  MoveL 3672 to (108.07, 245.49, -10) mm, rotated rx 180 ry 0 rz 180 deg; joints [-10.553, -45.82, 118.267, 168.944, 72.753, -176.684]
  MoveL 3673 to (108.64, 236.5, -10) mm, rotated rx -180 ry 0 rz 180 deg; joints [-10.17, -45.837, 118.333, 169.347, 72.78, -176.813]
  MoveL 3674 to (109.78, 227.56, -10) mm, rotated rx 180 ry 0 rz 180 deg; joints [-9.785, -45.844, 118.36, 169.751, 72.778, -176.936]
  MoveL 3675 to (111.49, 218.72, -10) mm, rotated rx -180 ry 0 rz -180 deg; joints [-9.4, -45.841, 118.347, 170.153, 72.749, -177.053]
  MoveL 3676 to (113.75, 209.99, -10) mm, rotated rx 180 ry 0 rz -180 deg; joints [-9.016, -45.827, 118.294, 170.552, 72.691, -177.166]
  MoveL 3677 to (116.56, 201.43, -10) mm, rotated rx 180 ry 0 rz -180 deg; joints [-8.636, -45.803, 118.202, 170.947, 72.605, -177.273]
  MoveL 3678 to (119.91, 193.07, -10) mm, rotated rx -180 ry 0 rz 180 deg; joints [-8.262, -45.769, 118.071, 171.334, 72.492, -177.375]
  MoveL 3679 to (123.79, 184.93, -10) mm, rotated rx 180 ry 0 rz 180 deg; joints [-7.896, -45.724, 117.902, 171.712, 72.352, -177.471]
  MoveL 3680 to (128.17, 177.06, -10) mm, rotated rx -180 ry 0 rz -180 deg; joints [-7.539, -45.669, 117.695, 172.079, 72.186, -177.563]
  MoveL 3681 to (133.04, 169.48, -10) mm, rotated rx 180 ry 0 rz 180 deg; joints [-7.194, -45.604, 117.451, 172.434, 71.995, -177.649]
  MoveL 3682 to (138.38, 162.22, -10) mm, rotated rx -180 ry 0 rz -180 deg; joints [-6.862, -45.529, 117.172, 172.774, 71.779, -177.73]
  MoveL 3683 to (144.17, 155.32, -10) mm, rotated rx -180 ry 0 rz -180 deg; joints [-6.544, -45.444, 116.858, 173.099, 71.54, -177.805]
  MoveL 3684 to (150.39, 148.8, -10) mm, rotated rx 180 ry 0 rz -180 deg; joints [-6.243, -45.349, 116.512, 173.406, 71.279, -177.875]
  MoveL 3685 to (157.01, 142.68, -10) mm, rotated rx 180 ry 0 rz 180 deg; joints [-5.96, -45.245, 116.135, 173.695, 70.998, -177.94]
  MoveL 3686 to (164, 137, -10) mm, rotated rx 180 ry 0 rz -180 deg; joints [-5.695, -45.131, 115.729, 173.964, 70.697, -177.998]
  MoveL 3687 to (171.34, 131.78, -10) mm, rotated rx 180 ry 0 rz -180 deg; joints [-5.45, -45.008, 115.294, 174.212, 70.379, -178.051]
  MoveL 3688 to (179, 127.02, -10) mm, rotated rx 180 ry 0 rz -180 deg; joints [-5.226, -44.877, 114.834, 174.439, 70.045, -178.097]
  MoveL 3689 to (186.94, 122.77, -10) mm, rotated rx -180 ry 0 rz -180 deg; joints [-5.024, -44.737, 114.351, 174.643, 69.696, -178.136]
  MoveL 3690 to (195.14, 119.03, -10) mm, rotated rx 180 ry 0 rz -180 deg; joints [-4.843, -44.589, 113.845, 174.823, 69.334, -178.169]
  MoveL 3691 to (203.56, 115.81, -10) mm, rotated rx 180 ry 0 rz -180 deg; joints [-4.685, -44.433, 113.321, 174.98, 68.961, -178.194]
  MoveL 3692 to (212.16, 113.13, -10) mm, rotated rx -180 ry 0 rz -180 deg; joints [-4.549, -44.271, 112.779, 175.112, 68.579, -178.211]
  MoveL 3693 to (220.92, 111.01, -10) mm, rotated rx -180 ry 0 rz -180 deg; joints [-4.437, -44.102, 112.222, 175.22, 68.189, -178.22]
  MoveL 3694 to (229.79, 109.45, -10) mm, rotated rx 180 ry 0 rz -180 deg; joints [-4.348, -43.927, 111.652, 175.303, 67.792, -178.221]
  MoveL 3695 to (238.75, 108.45, -10) mm, rotated rx -180 ry 0 rz 180 deg; joints [-4.282, -43.747, 111.072, 175.361, 67.392, -178.213]
  MoveL 3696 to (247.75, 108.02, -10) mm, rotated rx 180 ry 0 rz -180 deg; joints [-4.239, -43.563, 110.484, 175.394, 66.988, -178.196]
  MoveL 3697 to (256.76, 108.16, -10) mm, rotated rx -180 ry 0 rz -180 deg; joints [-4.218, -43.375, 109.891, 175.402, 66.584, -178.17]
  MoveL 3698 to (265.74, 108.87, -10) mm, rotated rx 180 ry 0 rz -180 deg; joints [-4.22, -43.183, 109.294, 175.386, 66.179, -178.133]
  MoveL 3699 to (274.66, 110.16, -10) mm, rotated rx 180 ry 0 rz 180 deg; joints [-4.244, -42.99, 108.697, 175.345, 65.778, -178.087]
  MoveL 3700 to (283.48, 112, -10) mm, rotated rx 180 ry 0 rz 180 deg; joints [-4.29, -42.795, 108.101, 175.28, 65.379, -178.03]
  MoveL 3701 to (292.16, 114.4, -10) mm, rotated rx 180 ry 0 rz 180 deg; joints [-4.356, -42.6, 107.508, 175.192, 64.986, -177.963]
  MoveL 3702 to (300.68, 117.35, -10) mm, rotated rx 180 ry 0 rz 180 deg; joints [-4.443, -42.405, 106.922, 175.081, 64.6, -177.886]
  MoveL 3703 to (308.99, 120.83, -10) mm, rotated rx 180 ry 0 rz 180 deg; joints [-4.549, -42.211, 106.345, 174.947, 64.222, -177.798]
  MoveL 3704 to (317.06, 124.83, -10) mm, rotated rx 180 ry 0 rz 180 deg; joints [-4.674, -42.019, 105.778, 174.791, 63.853, -177.7]
  MoveL 3705 to (324.87, 129.34, -10) mm, rotated rx -180 ry 0 rz 180 deg; joints [-4.818, -41.829, 105.224, 174.615, 63.495, -177.591]
  MoveL 3706 to (332.37, 134.33, -10) mm, rotated rx -180 ry 0 rz -180 deg; joints [-4.978, -41.644, 104.684, 174.418, 63.15, -177.473]
  MoveL 3707 to (339.54, 139.79, -10) mm, rotated rx -180 ry 0 rz 180 deg; joints [-5.156, -41.463, 104.162, 174.202, 62.818, -177.344]
  MoveL 3708 to (346.35, 145.69, -10) mm, rotated rx 180 ry 0 rz 180 deg; joints [-5.349, -41.288, 103.659, 173.968, 62.501, -177.206]
  MoveL 3709 to (352.77, 152.01, -10) mm, rotated rx -180 ry 0 rz 180 deg; joints [-5.557, -41.119, 103.176, 173.716, 62.2, -177.06]
  MoveL 3710 to (358.78, 158.72, -10) mm, rotated rx 180 ry 0 rz -180 deg; joints [-5.778, -40.957, 102.717, 173.447, 61.916, -176.905]
  MoveL 3711 to (364.35, 165.81, -10) mm, rotated rx 180 ry 0 rz -180 deg; joints [-6.013, -40.803, 102.282, 173.164, 61.65, -176.742]
  MoveL 3712 to (369.46, 173.23, -10) mm, rotated rx 180 ry 0 rz 180 deg; joints [-6.26, -40.657, 101.873, 172.866, 61.403, -176.572]
  MoveL 3713 to (374.09, 180.96, -10) mm, rotated rx 180 ry 0 rz 180 deg; joints [-6.518, -40.521, 101.491, 172.555, 61.176, -176.395]
  MoveL 3714 to (378.22, 188.97, -10) mm, rotated rx -180 ry 0 rz 180 deg; joints [-6.787, -40.394, 101.139, 172.233, 60.97, -176.213]
  MoveL 3715 to (381.83, 197.22, -10) mm, rotated rx 180 ry 0 rz -180 deg; joints [-7.064, -40.278, 100.818, 171.9, 60.785, -176.026]
  MoveL 3716 to (384.91, 205.69, -10) mm, rotated rx -180 ry 0 rz 180 deg; joints [-7.35, -40.174, 100.528, 171.558, 60.622, -175.836]
  MoveL 3717 to (387.45, 214.34, -10) mm, rotated rx 180 ry 0 rz 180 deg; joints [-7.643, -40.08, 100.271, 171.208, 60.482, -175.642]
  MoveL 3718 to (389.43, 223.13, -10) mm, rotated rx -180 ry 0 rz -180 deg; joints [-7.943, -39.999, 100.048, 170.852, 60.365, -175.447]
  MoveL 3719 to (390.86, 232.02, -10) mm, rotated rx -180 ry 0 rz -180 deg; joints [-8.248, -39.931, 99.86, 170.491, 60.272, -175.252]
  MoveL 3720 to (391.71, 240.99, -10) mm, rotated rx -180 ry 0 rz -180 deg; joints [-8.558, -39.875, 99.707, 170.126, 60.202, -175.056]
  MoveL 3721 to (392, 250, -10) mm, rotated rx 180 ry 0 rz -180 deg; joints [-8.871, -39.832, 99.591, 169.759, 60.157, -174.863]
  MoveL 3722 to (380, 250, -10) mm, rotated rx -180 ry 0 rz 180 deg; joints [-8.937, -40.137, 100.428, 169.737, 60.687, -174.934]
  MoveL 3723 to (379.74, 258.25, -10) mm, rotated rx 180 ry 0 rz 180 deg; joints [-9.229, -40.111, 100.355, 169.4, 60.667, -174.762]
  MoveL 3724 to (378.95, 266.46, -10) mm, rotated rx 180 ry 0 rz -180 deg; joints [-9.521, -40.096, 100.315, 169.063, 60.669, -174.592]
  MoveL 3725 to (377.65, 274.6, -10) mm, rotated rx 180 ry 0 rz 180 deg; joints [-9.815, -40.094, 100.309, 168.727, 60.694, -174.428]
  MoveL 3726 to (375.83, 282.65, -10) mm, rotated rx 180 ry 0 rz -180 deg; joints [-10.108, -40.104, 100.337, 168.395, 60.74, -174.268]
  MoveL 3727 to (373.51, 290.56, -10) mm, rotated rx -180 ry 0 rz -180 deg; joints [-10.4, -40.127, 100.399, 168.067, 60.808, -174.115]
  MoveL 3728 to (370.69, 298.32, -10) mm, rotated rx 180 ry 0 rz -180 deg; joints [-10.689, -40.161, 100.495, 167.744, 60.898, -173.969]
  MoveL 3729 to (367.38, 305.87, -10) mm, rotated rx 180 ry 0 rz 180 deg; joints [-10.976, -40.208, 100.623, 167.427, 61.009, -173.831]
  MoveL 3730 to (363.6, 313.21, -10) mm, rotated rx 180 ry 0 rz 180 deg; joints [-11.259, -40.266, 100.785, 167.119, 61.14, -173.701]
  MoveL 3731 to (359.36, 320.28, -10) mm, rotated rx 180 ry 0 rz 180 deg; joints [-11.537, -40.336, 100.978, 166.819, 61.291, -173.581]
  MoveL 3732 to (354.69, 327.08, -10) mm, rotated rx 180 ry 0 rz -180 deg; joints [-11.809, -40.417, 101.203, 166.529, 61.462, -173.471]
  MoveL 3733 to (349.59, 333.56, -10) mm, rotated rx -180 ry 0 rz -180 deg; joints [-12.075, -40.509, 101.458, 166.25, 61.651, -173.372]
  MoveL 3734 to (344.09, 339.71, -10) mm, rotated rx 180 ry 0 rz 180 deg; joints [-12.333, -40.611, 101.743, 165.982, 61.859, -173.284]
  MoveL 3735 to (338.21, 345.5, -10) mm, rotated rx -180 ry 0 rz 180 deg; joints [-12.582, -40.722, 102.056, 165.728, 62.083, -173.208]
  MoveL 3736 to (331.97, 350.9, -10) mm, rotated rx -180 ry 0 rz -180 deg; joints [-12.823, -40.843, 102.397, 165.487, 62.324, -173.144]
  MoveL 3737 to (325.41, 355.89, -10) mm, rotated rx 180 ry 0 rz 180 deg; joints [-13.053, -40.973, 102.763, 165.26, 62.581, -173.092]
  MoveL 3738 to (318.54, 360.46, -10) mm, rotated rx -180 ry 0 rz 180 deg; joints [-13.272, -41.111, 103.154, 165.049, 62.852, -173.053]
  MoveL 3739 to (311.4, 364.59, -10) mm, rotated rx 180 ry 0 rz -180 deg; joints [-13.479, -41.256, 103.567, 164.854, 63.136, -173.027]
  MoveL 3740 to (304, 368.25, -10) mm, rotated rx -180 ry 0 rz 180 deg; joints [-13.673, -41.408, 104.003, 164.675, 63.433, -173.013]
  MoveL 3741 to (296.4, 371.44, -10) mm, rotated rx -180 ry 0 rz -180 deg; joints [-13.854, -41.566, 104.457, 164.514, 63.742, -173.012]
  MoveL 3742 to (288.6, 374.14, -10) mm, rotated rx -180 ry 0 rz 180 deg; joints [-14.02, -41.729, 104.93, 164.371, 64.06, -173.023]
  MoveL 3743 to (280.65, 376.34, -10) mm, rotated rx -180 ry 0 rz -180 deg; joints [-14.172, -41.896, 105.419, 164.246, 64.388, -173.047]
  MoveL 3744 to (272.57, 378.03, -10) mm, rotated rx 180 ry 0 rz 180 deg; joints [-14.307, -42.068, 105.923, 164.14, 64.724, -173.084]
  MoveL 3745 to (264.41, 379.2, -10) mm, rotated rx 180 ry 0 rz -180 deg; joints [-14.426, -42.242, 106.439, 164.054, 65.067, -173.132]
  MoveL 3746 to (256.19, 379.85, -10) mm, rotated rx -180 ry 0 rz 180 deg; joints [-14.527, -42.419, 106.965, 163.987, 65.415, -173.191]
  MoveL 3747 to (247.94, 379.98, -10) mm, rotated rx -180 ry 0 rz 180 deg; joints [-14.611, -42.597, 107.499, 163.941, 65.767, -173.262]
  MoveL 3748 to (239.7, 379.59, -10) mm, rotated rx -180 ry 0 rz -180 deg; joints [-14.676, -42.775, 108.04, 163.915, 66.123, -173.343]
  MoveL 3749 to (231.5, 378.68, -10) mm, rotated rx -180 ry 0 rz -180 deg; joints [-14.722, -42.954, 108.585, 163.91, 66.48, -173.434]
  MoveL 3750 to (223.38, 377.24, -10) mm, rotated rx -180 ry 0 rz 180 deg; joints [-14.748, -43.131, 109.132, 163.926, 66.838, -173.534]
  MoveL 3751 to (215.36, 375.3, -10) mm, rotated rx -180 ry 0 rz -180 deg; joints [-14.754, -43.307, 109.679, 163.962, 67.196, -173.643]
  MoveL 3752 to (207.48, 372.85, -10) mm, rotated rx 180 ry 0 rz 180 deg; joints [-14.74, -43.48, 110.223, 164.02, 67.551, -173.759]
  MoveL 3753 to (199.78, 369.91, -10) mm, rotated rx -180 ry 0 rz -180 deg; joints [-14.705, -43.651, 110.763, 164.099, 67.903, -173.883]
  MoveL 3754 to (192.27, 366.48, -10) mm, rotated rx -180 ry 0 rz -180 deg; joints [-14.649, -43.817, 111.296, 164.199, 68.25, -174.014]
  MoveL 3755 to (185, 362.58, -10) mm, rotated rx 180 ry 0 rz -180 deg; joints [-14.573, -43.979, 111.821, 164.32, 68.59, -174.15]
  MoveL 3756 to (177.99, 358.23, -10) mm, rotated rx 180 ry 0 rz -180 deg; joints [-14.475, -44.136, 112.335, 164.462, 68.924, -174.29]
  MoveL 3757 to (171.27, 353.45, -10) mm, rotated rx -180 ry 0 rz -180 deg; joints [-14.356, -44.288, 112.835, 164.624, 69.249, -174.435]
  MoveL 3758 to (164.87, 348.25, -10) mm, rotated rx -180 ry 0 rz 180 deg; joints [-14.217, -44.433, 113.32, 164.806, 69.563, -174.583]
  MoveL 3759 to (158.81, 342.65, -10) mm, rotated rx -180 ry 0 rz -180 deg; joints [-14.057, -44.572, 113.789, 165.007, 69.866, -174.733]
  MoveL 3760 to (153.12, 336.68, -10) mm, rotated rx -180 ry 0 rz 180 deg; joints [-13.877, -44.704, 114.237, 165.228, 70.157, -174.885]
  MoveL 3761 to (147.81, 330.36, -10) mm, rotated rx 180 ry 0 rz 180 deg; joints [-13.677, -44.828, 114.665, 165.466, 70.433, -175.038]
  MoveL 3762 to (142.92, 323.72, -10) mm, rotated rx 180 ry 0 rz 180 deg; joints [-13.459, -44.944, 115.07, 165.722, 70.694, -175.191]
  MoveL 3763 to (138.46, 316.78, -10) mm, rotated rx 180 ry 0 rz 180 deg; joints [-13.223, -45.052, 115.45, 165.995, 70.938, -175.343]
  MoveL 3764 to (134.45, 309.57, -10) mm, rotated rx 180 ry 0 rz -180 deg; joints [-12.97, -45.152, 115.804, 166.283, 71.164, -175.494]
  MoveL 3765 to (130.91, 302.12, -10) mm, rotated rx -180 ry 0 rz -180 deg; joints [-12.7, -45.243, 116.13, 166.585, 71.371, -175.643]
  MoveL 3766 to (127.84, 294.46, -10) mm, rotated rx -180 ry 0 rz -180 deg; joints [-12.416, -45.325, 116.426, 166.901, 71.559, -175.79]
  MoveL 3767 to (125.27, 286.63, -10) mm, rotated rx -180 ry 0 rz -180 deg; joints [-12.118, -45.398, 116.691, 167.228, 71.725, -175.934]
  MoveL 3768 to (123.19, 278.64, -10) mm, rotated rx 180 ry 0 rz 180 deg; joints [-11.808, -45.462, 116.925, 167.566, 71.869, -176.075]
  MoveL 3769 to (121.63, 270.54, -10) mm, rotated rx 180 ry 0 rz -180 deg; joints [-11.487, -45.516, 117.125, 167.913, 71.99, -176.212]
  MoveL 3770 to (120.59, 262.36, -10) mm, rotated rx 180 ry 0 rz 180 deg; joints [-11.157, -45.561, 117.292, 168.267, 72.087, -176.345]
  MoveL 3771 to (120.07, 254.12, -10) mm, rotated rx 180 ry 0 rz 180 deg; joints [-10.819, -45.597, 117.423, 168.627, 72.161, -176.474]
  MoveL 3772 to (120.07, 245.88, -10) mm, rotated rx -180 ry 0 rz -180 deg; joints [-10.476, -45.622, 117.519, 168.992, 72.209, -176.598]
  MoveL 3773 to (120.59, 237.64, -10) mm, rotated rx 180 ry 0 rz -180 deg; joints [-10.128, -45.638, 117.58, 169.358, 72.232, -176.718]
  MoveL 3774 to (121.63, 229.46, -10) mm, rotated rx 180 ry 0 rz -180 deg; joints [-9.779, -45.645, 117.604, 169.726, 72.23, -176.834]
  MoveL 3775 to (123.19, 221.36, -10) mm, rotated rx 180 ry 0 rz 180 deg; joints [-9.429, -45.642, 117.592, 170.092, 72.203, -176.944]
  MoveL 3776 to (125.27, 213.37, -10) mm, rotated rx -180 ry 0 rz 180 deg; joints [-9.081, -45.629, 117.544, 170.455, 72.15, -177.05]
  MoveL 3777 to (127.84, 205.54, -10) mm, rotated rx -180 ry 0 rz -180 deg; joints [-8.736, -45.607, 117.46, 170.814, 72.072, -177.15]
  MoveL 3778 to (130.91, 197.88, -10) mm, rotated rx 180 ry 0 rz -180 deg; joints [-8.396, -45.574, 117.341, 171.166, 71.969, -177.246]
  MoveL 3779 to (134.45, 190.43, -10) mm, rotated rx -180 ry 0 rz -180 deg; joints [-8.064, -45.533, 117.186, 171.511, 71.841, -177.337]
  MoveL 3780 to (138.46, 183.22, -10) mm, rotated rx -180 ry 0 rz 180 deg; joints [-7.739, -45.482, 116.998, 171.845, 71.69, -177.422]
  MoveL 3781 to (142.92, 176.28, -10) mm, rotated rx 180 ry 0 rz 180 deg; joints [-7.425, -45.421, 116.776, 172.168, 71.516, -177.503]
  MoveL 3782 to (147.81, 169.64, -10) mm, rotated rx -180 ry 0 rz -180 deg; joints [-7.123, -45.351, 116.521, 172.479, 71.32, -177.579]
  MoveL 3783 to (153.12, 163.32, -10) mm, rotated rx 180 ry 0 rz 180 deg; joints [-6.834, -45.272, 116.235, 172.775, 71.103, -177.649]
  MoveL 3784 to (158.81, 157.35, -10) mm, rotated rx -180 ry 0 rz 180 deg; joints [-6.559, -45.185, 115.92, 173.056, 70.866, -177.714]
  MoveL 3785 to (164.87, 151.75, -10) mm, rotated rx -180 ry 0 rz 180 deg; joints [-6.3, -45.088, 115.575, 173.32, 70.61, -177.773]
  MoveL 3786 to (171.27, 146.55, -10) mm, rotated rx -180 ry 0 rz 180 deg; joints [-6.058, -44.983, 115.204, 173.566, 70.337, -177.827]
  MoveL 3787 to (177.99, 141.77, -10) mm, rotated rx 180 ry 0 rz 180 deg; joints [-5.833, -44.869, 114.808, 173.793, 70.047, -177.875]
  MoveL 3788 to (185, 137.42, -10) mm, rotated rx 180 ry 0 rz -180 deg; joints [-5.627, -44.747, 114.388, 174.001, 69.743, -177.916]
  MoveL 3789 to (192.27, 133.52, -10) mm, rotated rx -180 ry 0 rz 180 deg; joints [-5.44, -44.618, 113.946, 174.188, 69.425, -177.951]
  MoveL 3790 to (199.78, 130.09, -10) mm, rotated rx -180 ry 0 rz 180 deg; joints [-5.273, -44.482, 113.484, 174.354, 69.095, -177.98]
  MoveL 3791 to (207.48, 127.15, -10) mm, rotated rx 180 ry 0 rz 180 deg; joints [-5.127, -44.339, 113.004, 174.498, 68.755, -178.001]
  MoveL 3792 to (215.36, 124.7, -10) mm, rotated rx -180 ry 0 rz -180 deg; joints [-5.001, -44.189, 112.509, 174.62, 68.406, -178.015]
  MoveL 3793 to (223.38, 122.76, -10) mm, rotated rx 180 ry 0 rz 180 deg; joints [-4.896, -44.034, 112, 174.72, 68.05, -178.022]
  MoveL 3794 to (231.5, 121.32, -10) mm, rotated rx -180 ry 0 rz 180 deg; joints [-4.812, -43.874, 111.479, 174.798, 67.688, -178.02]
  MoveL 3795 to (239.7, 120.41, -10) mm, rotated rx 180 ry 0 rz 180 deg; joints [-4.749, -43.709, 110.948, 174.852, 67.322, -178.011]
  MoveL 3796 to (247.94, 120.02, -10) mm, rotated rx -180 ry 0 rz 180 deg; joints [-4.707, -43.539, 110.41, 174.884, 66.953, -177.993]
  MoveL 3797 to (256.19, 120.15, -10) mm, rotated rx 180 ry 0 rz -180 deg; joints [-4.686, -43.367, 109.867, 174.893, 66.583, -177.966]
  MoveL 3798 to (264.41, 120.8, -10) mm, rotated rx 180 ry 0 rz 180 deg; joints [-4.685, -43.192, 109.321, 174.879, 66.213, -177.93]
  MoveL 3799 to (272.57, 121.98, -10) mm, rotated rx -180 ry 0 rz 180 deg; joints [-4.704, -43.015, 108.774, 174.843, 65.845, -177.885]
  MoveL 3800 to (280.65, 123.66, -10) mm, rotated rx 180 ry 0 rz 180 deg; joints [-4.743, -42.837, 108.228, 174.785, 65.481, -177.831]
  MoveL 3801 to (288.6, 125.86, -10) mm, rotated rx -180 ry 0 rz -180 deg; joints [-4.802, -42.658, 107.685, 174.706, 65.121, -177.767]
  MoveL 3802 to (296.4, 128.56, -10) mm, rotated rx -180 ry 0 rz -180 deg; joints [-4.879, -42.48, 107.148, 174.605, 64.767, -177.694]
  MoveL 3803 to (304, 131.75, -10) mm, rotated rx -180 ry 0 rz 180 deg; joints [-4.974, -42.303, 106.619, 174.484, 64.42, -177.612]
  MoveL 3804 to (311.4, 135.41, -10) mm, rotated rx -180 ry 0 rz 180 deg; joints [-5.087, -42.128, 106.1, 174.342, 64.082, -177.521]
  MoveL 3805 to (318.54, 139.54, -10) mm, rotated rx 180 ry 0 rz 180 deg; joints [-5.217, -41.955, 105.592, 174.181, 63.754, -177.42]
  MoveL 3806 to (325.41, 144.11, -10) mm, rotated rx -180 ry 0 rz -180 deg; joints [-5.363, -41.786, 105.097, 174.002, 63.437, -177.31]
  MoveL 3807 to (331.97, 149.1, -10) mm, rotated rx 180 ry 0 rz 180 deg; joints [-5.524, -41.621, 104.619, 173.805, 63.133, -177.192]
  MoveL 3808 to (338.21, 154.5, -10) mm, rotated rx 180 ry 0 rz 180 deg; joints [-5.7, -41.462, 104.157, 173.591, 62.842, -177.065]
  MoveL 3809 to (344.09, 160.29, -10) mm, rotated rx 180 ry 0 rz -180 deg; joints [-5.89, -41.308, 103.715, 173.361, 62.566, -176.93]
  MoveL 3810 to (349.59, 166.44, -10) mm, rotated rx -180 ry 0 rz 180 deg; joints [-6.093, -41.16, 103.294, 173.115, 62.305, -176.788]
  MoveL 3811 to (354.69, 172.92, -10) mm, rotated rx -180 ry 0 rz 180 deg; joints [-6.308, -41.02, 102.895, 172.856, 62.06, -176.639]
  MoveL 3812 to (359.36, 179.72, -10) mm, rotated rx 180 ry 0 rz -180 deg; joints [-6.534, -40.887, 102.52, 172.584, 61.834, -176.484]
  MoveL 3813 to (363.6, 186.79, -10) mm, rotated rx -180 ry 0 rz -180 deg; joints [-6.771, -40.763, 102.171, 172.299, 61.625, -176.323]
  MoveL 3814 to (367.38, 194.13, -10) mm, rotated rx -180 ry 0 rz 180 deg; joints [-7.017, -40.648, 101.848, 172.004, 61.435, -176.158]
  MoveL 3815 to (370.69, 201.68, -10) mm, rotated rx -180 ry 0 rz -180 deg; joints [-7.273, -40.543, 101.553, 171.699, 61.265, -175.988]
  MoveL 3816 to (373.51, 209.44, -10) mm, rotated rx 180 ry 0 rz -180 deg; joints [-7.536, -40.448, 101.288, 171.386, 61.116, -175.815]
  MoveL 3817 to (375.83, 217.35, -10) mm, rotated rx 180 ry 0 rz 180 deg; joints [-7.806, -40.363, 101.052, 171.066, 60.987, -175.64]
  MoveL 3818 to (377.65, 225.4, -10) mm, rotated rx -180 ry 0 rz 180 deg; joints [-8.082, -40.289, 100.848, 170.739, 60.879, -175.463]
  MoveL 3819 to (378.95, 233.54, -10) mm, rotated rx -180 ry 0 rz -180 deg; joints [-8.363, -40.227, 100.675, 170.408, 60.793, -175.286]
  MoveL 3820 to (379.74, 241.75, -10) mm, rotated rx 180 ry 0 rz -180 deg; joints [-8.648, -40.176, 100.535, 170.074, 60.729, -175.109]
  MoveL 3821 to (380, 250, -10) mm, rotated rx -180 ry 0 rz 180 deg; joints [-8.937, -40.137, 100.428, 169.737, 60.687, -174.934]
  MoveL 3822 to (368, 250, -10) mm, rotated rx -180 ry 0 rz 180 deg; joints [-9.004, -40.438, 101.261, 169.714, 61.216, -175.006]
  MoveL 3823 to (367.76, 257.48, -10) mm, rotated rx 180 ry 0 rz 180 deg; joints [-9.27, -40.414, 101.194, 169.407, 61.198, -174.851]
  MoveL 3824 to (367.05, 264.94, -10) mm, rotated rx 180 ry 0 rz 180 deg; joints [-9.538, -40.401, 101.158, 169.1, 61.199, -174.7]
  MoveL 3825 to (365.87, 272.33, -10) mm, rotated rx 180 ry 0 rz 180 deg; joints [-9.806, -40.399, 101.153, 168.795, 61.221, -174.552]
  MoveL 3826 to (364.22, 279.64, -10) mm, rotated rx -180 ry 0 rz 180 deg; joints [-10.075, -40.408, 101.178, 168.492, 61.263, -174.409]
  MoveL 3827 to (362.11, 286.82, -10) mm, rotated rx 180 ry 0 rz -180 deg; joints [-10.341, -40.428, 101.234, 168.193, 61.325, -174.272]
  MoveL 3828 to (359.55, 293.86, -10) mm, rotated rx 180 ry 0 rz -180 deg; joints [-10.606, -40.46, 101.321, 167.899, 61.406, -174.141]
  MoveL 3829 to (356.55, 300.72, -10) mm, rotated rx -180 ry 0 rz 180 deg; joints [-10.868, -40.502, 101.438, 167.611, 61.506, -174.018]
  MoveL 3830 to (353.11, 307.37, -10) mm, rotated rx 180 ry 0 rz 180 deg; joints [-11.127, -40.554, 101.585, 167.33, 61.625, -173.902]
  MoveL 3831 to (349.27, 313.8, -10) mm, rotated rx 180 ry 0 rz 180 deg; joints [-11.381, -40.617, 101.761, 167.057, 61.763, -173.794]
  MoveL 3832 to (345.02, 319.96, -10) mm, rotated rx -180 ry 0 rz -180 deg; joints [-11.629, -40.69, 101.965, 166.793, 61.918, -173.696]
  MoveL 3833 to (340.39, 325.85, -10) mm, rotated rx 180 ry 0 rz 180 deg; joints [-11.871, -40.773, 102.197, 166.538, 62.09, -173.607]
  MoveL 3834 to (335.4, 331.43, -10) mm, rotated rx 180 ry 0 rz -180 deg; joints [-12.107, -40.865, 102.456, 166.295, 62.278, -173.528]
  MoveL 3835 to (330.06, 336.68, -10) mm, rotated rx 180 ry 0 rz 180 deg; joints [-12.334, -40.965, 102.741, 166.063, 62.483, -173.459]
  MoveL 3836 to (324.41, 341.59, -10) mm, rotated rx -180 ry 0 rz -180 deg; joints [-12.553, -41.074, 103.05, 165.843, 62.702, -173.401]
  MoveL 3837 to (318.45, 346.12, -10) mm, rotated rx -180 ry 0 rz 180 deg; joints [-12.762, -41.191, 103.383, 165.637, 62.936, -173.354]
  MoveL 3838 to (312.21, 350.27, -10) mm, rotated rx 180 ry 0 rz -180 deg; joints [-12.961, -41.316, 103.738, 165.445, 63.182, -173.319]
  MoveL 3839 to (305.73, 354.01, -10) mm, rotated rx -180 ry 0 rz -180 deg; joints [-13.149, -41.447, 104.114, 165.267, 63.441, -173.294]
  MoveL 3840 to (299.02, 357.34, -10) mm, rotated rx 180 ry 0 rz 180 deg; joints [-13.325, -41.584, 104.51, 165.104, 63.712, -173.281]
  MoveL 3841 to (292.11, 360.23, -10) mm, rotated rx 180 ry 0 rz 180 deg; joints [-13.488, -41.726, 104.923, 164.958, 63.992, -173.279]
  MoveL 3842 to (285.04, 362.68, -10) mm, rotated rx 180 ry 0 rz -180 deg; joints [-13.639, -41.874, 105.353, 164.828, 64.283, -173.289]
  MoveL 3843 to (277.82, 364.67, -10) mm, rotated rx 180 ry 0 rz 180 deg; joints [-13.775, -42.025, 105.797, 164.715, 64.581, -173.309]
  MoveL 3844 to (270.49, 366.21, -10) mm, rotated rx 180 ry 0 rz -180 deg; joints [-13.896, -42.18, 106.255, 164.619, 64.887, -173.341]
  MoveL 3845 to (263.08, 367.27, -10) mm, rotated rx 180 ry 0 rz -180 deg; joints [-14.002, -42.338, 106.723, 164.541, 65.199, -173.383]
  MoveL 3846 to (255.61, 367.87, -10) mm, rotated rx 180 ry 0 rz 180 deg; joints [-14.093, -42.498, 107.201, 164.481, 65.516, -173.435]
  MoveL 3847 to (248.13, 367.99, -10) mm, rotated rx -180 ry 0 rz -180 deg; joints [-14.167, -42.659, 107.687, 164.44, 65.837, -173.497]
  MoveL 3848 to (240.65, 367.63, -10) mm, rotated rx -180 ry 0 rz -180 deg; joints [-14.224, -42.821, 108.178, 164.418, 66.161, -173.569]
  MoveL 3849 to (233.21, 366.8, -10) mm, rotated rx -180 ry 0 rz -180 deg; joints [-14.263, -42.982, 108.673, 164.414, 66.486, -173.65]
  MoveL 3850 to (225.83, 365.5, -10) mm, rotated rx 180 ry 0 rz -180 deg; joints [-14.284, -43.143, 109.169, 164.43, 66.811, -173.739]
  MoveL 3851 to (218.56, 363.73, -10) mm, rotated rx -180 ry 0 rz 180 deg; joints [-14.288, -43.303, 109.666, 164.464, 67.136, -173.835]
  MoveL 3852 to (211.41, 361.51, -10) mm, rotated rx 180 ry 0 rz 180 deg; joints [-14.273, -43.46, 110.16, 164.519, 67.459, -173.939]
  MoveL 3853 to (204.41, 358.84, -10) mm, rotated rx -180 ry 0 rz -180 deg; joints [-14.239, -43.615, 110.65, 164.592, 67.779, -174.05]
  MoveL 3854 to (197.6, 355.73, -10) mm, rotated rx -180 ry 0 rz -180 deg; joints [-14.186, -43.766, 111.134, 164.684, 68.094, -174.166]
  MoveL 3855 to (191, 352.19, -10) mm, rotated rx 180 ry 0 rz 180 deg; joints [-14.114, -43.914, 111.609, 164.796, 68.403, -174.288]
  MoveL 3856 to (184.64, 348.24, -10) mm, rotated rx 180 ry 0 rz 180 deg; joints [-14.023, -44.057, 112.075, 164.926, 68.705, -174.414]
  MoveL 3857 to (178.54, 343.9, -10) mm, rotated rx -180 ry 0 rz -180 deg; joints [-13.913, -44.195, 112.529, 165.074, 69, -174.543]
  MoveL 3858 to (172.73, 339.18, -10) mm, rotated rx 180 ry 0 rz 180 deg; joints [-13.785, -44.328, 112.969, 165.241, 69.285, -174.676]
  MoveL 3859 to (167.23, 334.1, -10) mm, rotated rx 180 ry 0 rz 180 deg; joints [-13.639, -44.455, 113.393, 165.425, 69.559, -174.811]
  MoveL 3860 to (162.06, 328.68, -10) mm, rotated rx -180 ry 0 rz 180 deg; joints [-13.474, -44.575, 113.799, 165.626, 69.821, -174.948]
  MoveL 3861 to (157.25, 322.94, -10) mm, rotated rx 180 ry 0 rz -180 deg; joints [-13.292, -44.689, 114.187, 165.844, 70.071, -175.086]
  MoveL 3862 to (152.81, 316.91, -10) mm, rotated rx -180 ry 0 rz 180 deg; joints [-13.094, -44.796, 114.553, 166.077, 70.306, -175.224]
  MoveL 3863 to (148.76, 310.61, -10) mm, rotated rx -180 ry 0 rz 180 deg; joints [-12.879, -44.895, 114.897, 166.324, 70.526, -175.362]
  MoveL 3864 to (145.12, 304.07, -10) mm, rotated rx 180 ry 0 rz 180 deg; joints [-12.65, -44.986, 115.217, 166.586, 70.73, -175.5]
  MoveL 3865 to (141.9, 297.31, -10) mm, rotated rx 180 ry 0 rz 180 deg; joints [-12.406, -45.07, 115.512, 166.86, 70.917, -175.636]
  MoveL 3866 to (139.12, 290.36, -10) mm, rotated rx 180 ry 0 rz -180 deg; joints [-12.149, -45.145, 115.78, 167.146, 71.085, -175.77]
  MoveL 3867 to (136.78, 283.24, -10) mm, rotated rx 180 ry 0 rz 180 deg; joints [-11.879, -45.213, 116.02, 167.443, 71.234, -175.901]
  MoveL 3868 to (134.9, 276, -10) mm, rotated rx -180 ry 0 rz -180 deg; joints [-11.6, -45.271, 116.231, 167.749, 71.363, -176.03]
  MoveL 3869 to (133.48, 268.64, -10) mm, rotated rx 180 ry 0 rz 180 deg; joints [-11.31, -45.321, 116.412, 168.063, 71.471, -176.156]
  MoveL 3870 to (132.53, 261.22, -10) mm, rotated rx -180 ry 0 rz 180 deg; joints [-11.013, -45.363, 116.563, 168.383, 71.559, -176.279]
  MoveL 3871 to (132.06, 253.74, -10) mm, rotated rx 180 ry 0 rz -180 deg; joints [-10.709, -45.396, 116.682, 168.708, 71.624, -176.398]
  MoveL 3872 to (132.06, 246.26, -10) mm, rotated rx 180 ry 0 rz 180 deg; joints [-10.4, -45.419, 116.769, 169.037, 71.667, -176.513]
  MoveL 3873 to (132.53, 238.78, -10) mm, rotated rx -180 ry 0 rz -180 deg; joints [-10.087, -45.434, 116.823, 169.368, 71.687, -176.624]
  MoveL 3874 to (133.48, 231.36, -10) mm, rotated rx 180 ry 0 rz 180 deg; joints [-9.773, -45.44, 116.845, 169.7, 71.684, -176.731]
  MoveL 3875 to (134.9, 224, -10) mm, rotated rx -180 ry 0 rz -180 deg; joints [-9.458, -45.437, 116.835, 170.03, 71.659, -176.834]
  MoveL 3876 to (136.78, 216.76, -10) mm, rotated rx 180 ry 0 rz -180 deg; joints [-9.145, -45.426, 116.791, 170.358, 71.611, -176.932]
  MoveL 3877 to (139.12, 209.64, -10) mm, rotated rx -180 ry 0 rz -180 deg; joints [-8.835, -45.405, 116.715, 170.682, 71.54, -177.026]
  MoveL 3878 to (141.9, 202.69, -10) mm, rotated rx 180 ry 0 rz 180 deg; joints [-8.529, -45.375, 116.607, 171, 71.447, -177.115]
  MoveL 3879 to (145.12, 195.93, -10) mm, rotated rx 180 ry 0 rz 180 deg; joints [-8.229, -45.337, 116.468, 171.311, 71.332, -177.199]
  MoveL 3880 to (148.76, 189.39, -10) mm, rotated rx -180 ry 0 rz -180 deg; joints [-7.937, -45.29, 116.297, 171.613, 71.196, -177.279]
  MoveL 3881 to (152.81, 183.09, -10) mm, rotated rx -180 ry 0 rz -180 deg; joints [-7.653, -45.234, 116.096, 171.905, 71.039, -177.354]
  MoveL 3882 to (157.25, 177.06, -10) mm, rotated rx -180 ry 0 rz -180 deg; joints [-7.38, -45.17, 115.866, 172.185, 70.863, -177.424]
  MoveL 3883 to (162.06, 171.32, -10) mm, rotated rx 180 ry 0 rz -180 deg; joints [-7.119, -45.097, 115.608, 172.453, 70.667, -177.489]
  MoveL 3884 to (167.23, 165.9, -10) mm, rotated rx -180 ry 0 rz -180 deg; joints [-6.87, -45.016, 115.322, 172.707, 70.453, -177.548]
  MoveL 3885 to (172.73, 160.82, -10) mm, rotated rx -180 ry 0 rz 180 deg; joints [-6.636, -44.927, 115.011, 172.946, 70.222, -177.603]
  MoveL 3886 to (178.54, 156.1, -10) mm, rotated rx -180 ry 0 rz 180 deg; joints [-6.416, -44.831, 114.675, 173.17, 69.976, -177.651]
  MoveL 3887 to (184.64, 151.76, -10) mm, rotated rx -180 ry 0 rz 180 deg; joints [-6.212, -44.727, 114.316, 173.376, 69.714, -177.694]
  MoveL 3888 to (191, 147.81, -10) mm, rotated rx 180 ry 0 rz 180 deg; joints [-6.024, -44.615, 113.935, 173.565, 69.439, -177.732]
  MoveL 3889 to (197.6, 144.27, -10) mm, rotated rx 180 ry 0 rz 180 deg; joints [-5.853, -44.497, 113.535, 173.735, 69.152, -177.763]
  MoveL 3890 to (204.41, 141.16, -10) mm, rotated rx 180 ry 0 rz 180 deg; joints [-5.701, -44.372, 113.117, 173.886, 68.855, -177.787]
  MoveL 3891 to (211.41, 138.49, -10) mm, rotated rx 180 ry 0 rz -180 deg; joints [-5.566, -44.242, 112.682, 174.018, 68.547, -177.805]
  MoveL 3892 to (218.56, 136.27, -10) mm, rotated rx 180 ry 0 rz 180 deg; joints [-5.45, -44.105, 112.233, 174.13, 68.232, -177.817]
  MoveL 3893 to (225.83, 134.5, -10) mm, rotated rx 180 ry 0 rz -180 deg; joints [-5.353, -43.964, 111.771, 174.222, 67.909, -177.821]
  MoveL 3894 to (233.21, 133.2, -10) mm, rotated rx 180 ry 0 rz 180 deg; joints [-5.274, -43.818, 111.299, 174.293, 67.582, -177.817]
  MoveL 3895 to (240.65, 132.37, -10) mm, rotated rx 180 ry 0 rz -180 deg; joints [-5.215, -43.668, 110.818, 174.344, 67.25, -177.807]
  MoveL 3896 to (248.13, 132.01, -10) mm, rotated rx -180 ry 0 rz -180 deg; joints [-5.174, -43.514, 110.33, 174.374, 66.916, -177.788]
  MoveL 3897 to (255.61, 132.13, -10) mm, rotated rx 180 ry 0 rz 180 deg; joints [-5.153, -43.357, 109.837, 174.383, 66.58, -177.761]
  MoveL 3898 to (263.08, 132.73, -10) mm, rotated rx 180 ry 0 rz 180 deg; joints [-5.15, -43.198, 109.341, 174.372, 66.245, -177.727]
  MoveL 3899 to (270.49, 133.79, -10) mm, rotated rx 180 ry 0 rz -180 deg; joints [-5.165, -43.038, 108.844, 174.341, 65.911, -177.684]
  MoveL 3900 to (277.82, 135.33, -10) mm, rotated rx 180 ry 0 rz -180 deg; joints [-5.198, -42.876, 108.348, 174.289, 65.58, -177.633]
  MoveL 3901 to (285.04, 137.32, -10) mm, rotated rx -180 ry 0 rz -180 deg; joints [-5.249, -42.715, 107.856, 174.218, 65.253, -177.573]
  MoveL 3902 to (292.11, 139.77, -10) mm, rotated rx 180 ry 0 rz 180 deg; joints [-5.317, -42.553, 107.368, 174.128, 64.931, -177.505]
  MoveL 3903 to (299.02, 142.66, -10) mm, rotated rx 180 ry 0 rz 180 deg; joints [-5.402, -42.393, 106.887, 174.019, 64.616, -177.428]
  MoveL 3904 to (305.73, 145.99, -10) mm, rotated rx -180 ry 0 rz -180 deg; joints [-5.503, -42.234, 106.415, 173.892, 64.309, -177.344]
  MoveL 3905 to (312.21, 149.73, -10) mm, rotated rx 180 ry 0 rz 180 deg; joints [-5.619, -42.078, 105.954, 173.747, 64.01, -177.251]
  MoveL 3906 to (318.45, 153.88, -10) mm, rotated rx 180 ry 0 rz -180 deg; joints [-5.75, -41.926, 105.505, 173.585, 63.722, -177.15]
  MoveL 3907 to (324.41, 158.41, -10) mm, rotated rx -180 ry 0 rz -180 deg; joints [-5.896, -41.777, 105.07, 173.406, 63.445, -177.042]
  MoveL 3908 to (330.06, 163.32, -10) mm, rotated rx -180 ry 0 rz -180 deg; joints [-6.055, -41.632, 104.65, 173.212, 63.181, -176.926]
  MoveL 3909 to (335.4, 168.57, -10) mm, rotated rx -180 ry 0 rz 180 deg; joints [-6.226, -41.493, 104.249, 173.004, 62.929, -176.804]
  MoveL 3910 to (340.39, 174.15, -10) mm, rotated rx 180 ry 0 rz 180 deg; joints [-6.41, -41.36, 103.866, 172.782, 62.692, -176.675]
  MoveL 3911 to (345.02, 180.04, -10) mm, rotated rx -180 ry 0 rz 180 deg; joints [-6.605, -41.234, 103.503, 172.547, 62.469, -176.539]
  MoveL 3912 to (349.27, 186.2, -10) mm, rotated rx -180 ry 0 rz 180 deg; joints [-6.811, -41.114, 103.162, 172.299, 62.263, -176.399]
  MoveL 3913 to (353.11, 192.63, -10) mm, rotated rx -180 ry 0 rz 180 deg; joints [-7.027, -41.002, 102.845, 172.041, 62.073, -176.254]
  MoveL 3914 to (356.55, 199.28, -10) mm, rotated rx 180 ry 0 rz 180 deg; joints [-7.251, -40.898, 102.551, 171.774, 61.9, -176.104]
  MoveL 3915 to (359.55, 206.14, -10) mm, rotated rx 180 ry 0 rz -180 deg; joints [-7.484, -40.803, 102.283, 171.497, 61.745, -175.952]
  MoveL 3916 to (362.11, 213.18, -10) mm, rotated rx -180 ry 0 rz -180 deg; joints [-7.724, -40.717, 102.042, 171.212, 61.609, -175.796]
  MoveL 3917 to (364.22, 220.36, -10) mm, rotated rx -180 ry 0 rz -180 deg; joints [-7.97, -40.641, 101.828, 170.921, 61.491, -175.639]
  MoveL 3918 to (365.87, 227.67, -10) mm, rotated rx -180 ry 0 rz -180 deg; joints [-8.222, -40.575, 101.642, 170.625, 61.393, -175.48]
  MoveL 3919 to (367.05, 235.06, -10) mm, rotated rx 180 ry 0 rz 180 deg; joints [-8.479, -40.519, 101.485, 170.324, 61.314, -175.321]
  MoveL 3920 to (367.76, 242.52, -10) mm, rotated rx -180 ry 0 rz -180 deg; joints [-8.74, -40.473, 101.358, 170.02, 61.255, -175.163]
  MoveL 3921 to (368, 250, -10) mm, rotated rx -180 ry 0 rz 180 deg; joints [-9.004, -40.438, 101.261, 169.714, 61.216, -175.006]
  MoveL 3922 to (356, 250, -10) mm, rotated rx -180 ry 0 rz 180 deg; joints [-9.072, -40.734, 102.088, 169.688, 61.745, -175.077]
  MoveL 3923 to (355.79, 256.72, -10) mm, rotated rx 180 ry 0 rz -180 deg; joints [-9.313, -40.713, 102.028, 169.412, 61.728, -174.94]
  MoveL 3924 to (355.15, 263.42, -10) mm, rotated rx -180 ry 0 rz 180 deg; joints [-9.555, -40.701, 101.996, 169.136, 61.729, -174.806]
  MoveL 3925 to (354.08, 270.06, -10) mm, rotated rx -180 ry 0 rz 180 deg; joints [-9.798, -40.699, 101.991, 168.861, 61.748, -174.675]
  MoveL 3926 to (352.6, 276.62, -10) mm, rotated rx 180 ry 0 rz -180 deg; joints [-10.041, -40.707, 102.014, 168.588, 61.786, -174.549]
  MoveL 3927 to (350.71, 283.08, -10) mm, rotated rx 180 ry 0 rz -180 deg; joints [-10.282, -40.725, 102.064, 168.319, 61.841, -174.427]
  MoveL 3928 to (348.41, 289.4, -10) mm, rotated rx 180 ry 0 rz -180 deg; joints [-10.522, -40.753, 102.143, 168.054, 61.914, -174.312]
  MoveL 3929 to (345.71, 295.56, -10) mm, rotated rx 180 ry 0 rz 180 deg; joints [-10.759, -40.791, 102.248, 167.794, 62.004, -174.202]
  MoveL 3930 to (342.63, 301.54, -10) mm, rotated rx -180 ry 0 rz -180 deg; joints [-10.993, -40.838, 102.38, 167.541, 62.111, -174.099]
  MoveL 3931 to (339.17, 307.31, -10) mm, rotated rx -180 ry 0 rz -180 deg; joints [-11.222, -40.894, 102.538, 167.295, 62.234, -174.004]
  MoveL 3932 to (335.36, 312.85, -10) mm, rotated rx -180 ry 0 rz -180 deg; joints [-11.447, -40.959, 102.722, 167.056, 62.373, -173.917]
  MoveL 3933 to (331.2, 318.14, -10) mm, rotated rx -180 ry 0 rz -180 deg; joints [-11.665, -41.032, 102.931, 166.827, 62.528, -173.838]
  MoveL 3934 to (326.72, 323.15, -10) mm, rotated rx 180 ry 0 rz 180 deg; joints [-11.878, -41.114, 103.164, 166.607, 62.698, -173.767]
  MoveL 3935 to (321.92, 327.87, -10) mm, rotated rx 180 ry 0 rz 180 deg; joints [-12.083, -41.204, 103.42, 166.398, 62.882, -173.706]
  MoveL 3936 to (316.84, 332.27, -10) mm, rotated rx -180 ry 0 rz -180 deg; joints [-12.28, -41.302, 103.698, 166.2, 63.08, -173.654]
  MoveL 3937 to (311.49, 336.35, -10) mm, rotated rx 180 ry 0 rz 180 deg; joints [-12.468, -41.406, 103.998, 166.014, 63.29, -173.612]
  MoveL 3938 to (305.89, 340.07, -10) mm, rotated rx -180 ry 0 rz -180 deg; joints [-12.647, -41.517, 104.317, 165.841, 63.512, -173.58]
  MoveL 3939 to (300.06, 343.43, -10) mm, rotated rx 180 ry 0 rz -180 deg; joints [-12.815, -41.634, 104.655, 165.681, 63.746, -173.558]
  MoveL 3940 to (294.03, 346.42, -10) mm, rotated rx -180 ry 0 rz 180 deg; joints [-12.973, -41.757, 105.011, 165.535, 63.989, -173.545]
  MoveL 3941 to (287.83, 349.02, -10) mm, rotated rx 180 ry 0 rz 180 deg; joints [-13.119, -41.884, 105.383, 165.403, 64.242, -173.543]
  MoveL 3942 to (281.47, 351.22, -10) mm, rotated rx 180 ry 0 rz -180 deg; joints [-13.253, -42.016, 105.77, 165.286, 64.504, -173.551]
  MoveL 3943 to (274.99, 353.01, -10) mm, rotated rx 180 ry 0 rz 180 deg; joints [-13.375, -42.151, 106.169, 165.185, 64.773, -173.568]
  MoveL 3944 to (268.41, 354.39, -10) mm, rotated rx -180 ry 0 rz 180 deg; joints [-13.483, -42.29, 106.581, 165.099, 65.049, -173.595]
  MoveL 3945 to (261.75, 355.35, -10) mm, rotated rx 180 ry 0 rz -180 deg; joints [-13.577, -42.431, 107.002, 165.029, 65.33, -173.631]
  MoveL 3946 to (255.04, 355.88, -10) mm, rotated rx -180 ry 0 rz 180 deg; joints [-13.656, -42.574, 107.432, 164.976, 65.615, -173.677]
  MoveL 3947 to (248.32, 355.99, -10) mm, rotated rx 180 ry 0 rz -180 deg; joints [-13.721, -42.719, 107.868, 164.94, 65.904, -173.731]
  MoveL 3948 to (241.6, 355.67, -10) mm, rotated rx -180 ry 0 rz 180 deg; joints [-13.77, -42.864, 108.31, 164.921, 66.196, -173.794]
  MoveL 3949 to (234.91, 354.92, -10) mm, rotated rx 180 ry 0 rz -180 deg; joints [-13.803, -43.009, 108.754, 164.919, 66.489, -173.864]
  MoveL 3950 to (228.29, 353.75, -10) mm, rotated rx 180 ry 0 rz -180 deg; joints [-13.821, -43.153, 109.2, 164.934, 66.782, -173.942]
  MoveL 3951 to (221.75, 352.17, -10) mm, rotated rx -180 ry 0 rz 180 deg; joints [-13.821, -43.297, 109.646, 164.966, 67.074, -174.027]
  MoveL 3952 to (215.33, 350.17, -10) mm, rotated rx -180 ry 0 rz 180 deg; joints [-13.806, -43.438, 110.09, 165.016, 67.365, -174.119]
  MoveL 3953 to (209.05, 347.77, -10) mm, rotated rx -180 ry 0 rz -180 deg; joints [-13.773, -43.577, 110.53, 165.084, 67.652, -174.216]
  MoveL 3954 to (202.93, 344.98, -10) mm, rotated rx -180 ry 0 rz -180 deg; joints [-13.723, -43.714, 110.964, 165.168, 67.935, -174.319]
  MoveL 3955 to (197, 341.8, -10) mm, rotated rx 180 ry 0 rz -180 deg; joints [-13.657, -43.847, 111.391, 165.27, 68.213, -174.427]
  MoveL 3956 to (191.28, 338.25, -10) mm, rotated rx 180 ry 0 rz -180 deg; joints [-13.574, -43.976, 111.809, 165.388, 68.484, -174.538]
  MoveL 3957 to (185.81, 334.35, -10) mm, rotated rx 180 ry 0 rz -180 deg; joints [-13.474, -44.1, 112.216, 165.523, 68.748, -174.653]
  MoveL 3958 to (180.58, 330.11, -10) mm, rotated rx -180 ry 0 rz -180 deg; joints [-13.357, -44.22, 112.611, 165.673, 69.003, -174.771]
  MoveL 3959 to (175.64, 325.55, -10) mm, rotated rx 180 ry 0 rz -180 deg; joints [-13.224, -44.335, 112.991, 165.84, 69.249, -174.892]
  MoveL 3960 to (171, 320.68, -10) mm, rotated rx 180 ry 0 rz 180 deg; joints [-13.076, -44.444, 113.356, 166.022, 69.484, -175.014]
  MoveL 3961 to (166.68, 315.52, -10) mm, rotated rx -180 ry 0 rz 180 deg; joints [-12.912, -44.547, 113.703, 166.218, 69.707, -175.137]
  MoveL 3962 to (162.69, 310.11, -10) mm, rotated rx -180 ry 0 rz 180 deg; joints [-12.733, -44.643, 114.031, 166.428, 69.917, -175.261]
  MoveL 3963 to (159.05, 304.45, -10) mm, rotated rx 180 ry 0 rz -180 deg; joints [-12.54, -44.733, 114.339, 166.65, 70.113, -175.385]
  MoveL 3964 to (155.78, 298.57, -10) mm, rotated rx 180 ry 0 rz 180 deg; joints [-12.334, -44.817, 114.626, 166.886, 70.295, -175.508]
  MoveL 3965 to (152.89, 292.5, -10) mm, rotated rx 180 ry 0 rz 180 deg; joints [-12.115, -44.893, 114.89, 167.132, 70.461, -175.631]
  MoveL 3966 to (150.39, 286.25, -10) mm, rotated rx -180 ry 0 rz 180 deg; joints [-11.885, -44.961, 115.13, 167.389, 70.611, -175.752]
  MoveL 3967 to (148.29, 279.86, -10) mm, rotated rx 180 ry 0 rz -180 deg; joints [-11.645, -45.022, 115.345, 167.654, 70.743, -175.871]
  MoveL 3968 to (146.6, 273.35, -10) mm, rotated rx 180 ry 0 rz -180 deg; joints [-11.395, -45.076, 115.533, 167.928, 70.858, -175.989]
  MoveL 3969 to (145.33, 266.75, -10) mm, rotated rx -180 ry 0 rz 180 deg; joints [-11.137, -45.122, 115.695, 168.209, 70.954, -176.103]
  MoveL 3970 to (144.48, 260.08, -10) mm, rotated rx 180 ry 0 rz -180 deg; joints [-10.872, -45.159, 115.83, 168.496, 71.031, -176.215]
  MoveL 3971 to (144.05, 253.36, -10) mm, rotated rx -180 ry 0 rz 180 deg; joints [-10.601, -45.189, 115.936, 168.787, 71.088, -176.324]
  MoveL 3972 to (144.05, 246.64, -10) mm, rotated rx -180 ry 0 rz 180 deg; joints [-10.325, -45.211, 116.014, 169.081, 71.126, -176.429]
  MoveL 3973 to (144.48, 239.92, -10) mm, rotated rx -180 ry 0 rz -180 deg; joints [-10.047, -45.225, 116.063, 169.377, 71.144, -176.531]
  MoveL 3974 to (145.33, 233.25, -10) mm, rotated rx -180 ry 0 rz -180 deg; joints [-9.767, -45.23, 116.083, 169.673, 71.141, -176.629]
  MoveL 3975 to (146.6, 226.65, -10) mm, rotated rx 180 ry 0 rz -180 deg; joints [-9.487, -45.227, 116.073, 169.968, 71.118, -176.723]
  MoveL 3976 to (148.29, 220.14, -10) mm, rotated rx 180 ry 0 rz 180 deg; joints [-9.208, -45.217, 116.034, 170.261, 71.074, -176.814]
  MoveL 3977 to (150.39, 213.75, -10) mm, rotated rx -180 ry 0 rz 180 deg; joints [-8.931, -45.198, 115.967, 170.55, 71.011, -176.9]
  MoveL 3978 to (152.89, 207.5, -10) mm, rotated rx -180 ry 0 rz 180 deg; joints [-8.659, -45.171, 115.87, 170.834, 70.928, -176.982]
  MoveL 3979 to (155.78, 201.43, -10) mm, rotated rx 180 ry 0 rz -180 deg; joints [-8.391, -45.136, 115.745, 171.112, 70.825, -177.06]
  MoveL 3980 to (159.05, 195.55, -10) mm, rotated rx 180 ry 0 rz 180 deg; joints [-8.131, -45.093, 115.592, 171.382, 70.704, -177.133]
  MoveL 3981 to (162.69, 189.89, -10) mm, rotated rx 180 ry 0 rz 180 deg; joints [-7.878, -45.042, 115.413, 171.643, 70.564, -177.201]
  MoveL 3982 to (166.68, 184.48, -10) mm, rotated rx -180 ry 0 rz -180 deg; joints [-7.634, -44.983, 115.207, 171.894, 70.406, -177.265]
  MoveL 3983 to (171, 179.32, -10) mm, rotated rx 180 ry 0 rz 180 deg; joints [-7.4, -44.917, 114.975, 172.134, 70.231, -177.325]
  MoveL 3984 to (175.64, 174.45, -10) mm, rotated rx -180 ry 0 rz 180 deg; joints [-7.177, -44.844, 114.72, 172.361, 70.04, -177.379]
  MoveL 3985 to (180.58, 169.89, -10) mm, rotated rx -180 ry 0 rz 180 deg; joints [-6.967, -44.763, 114.441, 172.576, 69.834, -177.428]
  MoveL 3986 to (185.81, 165.65, -10) mm, rotated rx 180 ry 0 rz 180 deg; joints [-6.769, -44.675, 114.14, 172.776, 69.614, -177.472]
  MoveL 3987 to (191.28, 161.75, -10) mm, rotated rx 180 ry 0 rz 180 deg; joints [-6.586, -44.581, 113.818, 172.961, 69.381, -177.51]
  MoveL 3988 to (197, 158.2, -10) mm, rotated rx -180 ry 0 rz -180 deg; joints [-6.417, -44.48, 113.478, 173.131, 69.135, -177.543]
  MoveL 3989 to (202.93, 155.02, -10) mm, rotated rx -180 ry 0 rz 180 deg; joints [-6.263, -44.373, 113.119, 173.284, 68.879, -177.57]
  MoveL 3990 to (209.05, 152.23, -10) mm, rotated rx 180 ry 0 rz -180 deg; joints [-6.124, -44.26, 112.744, 173.421, 68.612, -177.592]
  MoveL 3991 to (215.33, 149.83, -10) mm, rotated rx -180 ry 0 rz -180 deg; joints [-6.002, -44.142, 112.354, 173.54, 68.337, -177.607]
  MoveL 3992 to (221.75, 147.83, -10) mm, rotated rx 180 ry 0 rz 180 deg; joints [-5.896, -44.019, 111.951, 173.641, 68.055, -177.615]
  MoveL 3993 to (228.29, 146.25, -10) mm, rotated rx 180 ry 0 rz 180 deg; joints [-5.807, -43.892, 111.537, 173.725, 67.766, -177.617]
  MoveL 3994 to (234.91, 145.08, -10) mm, rotated rx 180 ry 0 rz 180 deg; joints [-5.735, -43.76, 111.113, 173.79, 67.472, -177.613]
  MoveL 3995 to (241.6, 144.33, -10) mm, rotated rx -180 ry 0 rz 180 deg; joints [-5.679, -43.625, 110.681, 173.836, 67.175, -177.601]
  MoveL 3996 to (248.32, 144.01, -10) mm, rotated rx 180 ry 0 rz 180 deg; joints [-5.641, -43.486, 110.243, 173.864, 66.875, -177.582]
  MoveL 3997 to (255.04, 144.12, -10) mm, rotated rx 180 ry 0 rz -180 deg; joints [-5.619, -43.346, 109.8, 173.874, 66.574, -177.557]
  MoveL 3998 to (261.75, 144.65, -10) mm, rotated rx 180 ry 0 rz 180 deg; joints [-5.615, -43.203, 109.354, 173.865, 66.273, -177.524]
  MoveL 3999 to (268.41, 145.61, -10) mm, rotated rx 180 ry 0 rz 180 deg; joints [-5.626, -43.059, 108.908, 173.838, 65.973, -177.483]
  MoveL 4000 to (274.99, 146.99, -10) mm, rotated rx 180 ry 0 rz 180 deg; joints [-5.654, -42.914, 108.463, 173.793, 65.676, -177.435]
  MoveL 4001 to (281.47, 148.78, -10) mm, rotated rx 180 ry 0 rz -180 deg; joints [-5.698, -42.769, 108.02, 173.73, 65.382, -177.38]
  MoveL 4002 to (287.83, 150.98, -10) mm, rotated rx 180 ry 0 rz -180 deg; joints [-5.757, -42.624, 107.582, 173.65, 65.093, -177.317]
  MoveL 4003 to (294.03, 153.58, -10) mm, rotated rx 180 ry 0 rz 180 deg; joints [-5.831, -42.48, 107.149, 173.553, 64.809, -177.246]
  MoveL 4004 to (300.06, 156.57, -10) mm, rotated rx 180 ry 0 rz -180 deg; joints [-5.921, -42.338, 106.725, 173.44, 64.533, -177.169]
  MoveL 4005 to (305.89, 159.93, -10) mm, rotated rx 180 ry 0 rz 180 deg; joints [-6.024, -42.199, 106.31, 173.31, 64.265, -177.084]
  MoveL 4006 to (311.49, 163.65, -10) mm, rotated rx 180 ry 0 rz -180 deg; joints [-6.14, -42.062, 105.906, 173.165, 64.005, -176.993]
  MoveL 4007 to (316.84, 167.73, -10) mm, rotated rx -180 ry 0 rz -180 deg; joints [-6.27, -41.929, 105.515, 173.006, 63.756, -176.895]
  MoveL 4008 to (321.92, 172.13, -10) mm, rotated rx 180 ry 0 rz 180 deg; joints [-6.412, -41.8, 105.138, 172.832, 63.518, -176.79]
  MoveL 4009 to (326.72, 176.85, -10) mm, rotated rx 180 ry 0 rz 180 deg; joints [-6.566, -41.676, 104.776, 172.645, 63.291, -176.68]
  MoveL 4010 to (331.2, 181.86, -10) mm, rotated rx 180 ry 0 rz 180 deg; joints [-6.731, -41.557, 104.432, 172.446, 63.077, -176.564]
  MoveL 4011 to (335.36, 187.15, -10) mm, rotated rx 180 ry 0 rz -180 deg; joints [-6.907, -41.444, 104.106, 172.235, 62.877, -176.443]
  MoveL 4012 to (339.17, 192.69, -10) mm, rotated rx -180 ry 0 rz 180 deg; joints [-7.092, -41.337, 103.799, 172.013, 62.69, -176.317]
  MoveL 4013 to (342.63, 198.46, -10) mm, rotated rx -180 ry 0 rz 180 deg; joints [-7.286, -41.237, 103.513, 171.782, 62.519, -176.187]
  MoveL 4014 to (345.71, 204.44, -10) mm, rotated rx 180 ry 0 rz 180 deg; joints [-7.488, -41.145, 103.249, 171.541, 62.363, -176.054]
  MoveL 4015 to (348.41, 210.6, -10) mm, rotated rx -180 ry 0 rz -180 deg; joints [-7.698, -41.06, 103.008, 171.292, 62.223, -175.917]
  MoveL 4016 to (350.71, 216.92, -10) mm, rotated rx 180 ry 0 rz 180 deg; joints [-7.914, -40.983, 102.791, 171.037, 62.1, -175.779]
  MoveL 4017 to (352.6, 223.38, -10) mm, rotated rx 180 ry 0 rz 180 deg; joints [-8.137, -40.915, 102.599, 170.775, 61.994, -175.639]
  MoveL 4018 to (354.08, 229.94, -10) mm, rotated rx -180 ry 0 rz 180 deg; joints [-8.365, -40.856, 102.431, 170.508, 61.905, -175.498]
  MoveL 4019 to (355.15, 236.58, -10) mm, rotated rx 180 ry 0 rz 180 deg; joints [-8.597, -40.806, 102.29, 170.237, 61.834, -175.357]
  MoveL 4020 to (355.79, 243.28, -10) mm, rotated rx -180 ry 0 rz -180 deg; joints [-8.833, -40.765, 102.176, 169.964, 61.78, -175.216]
  MoveL 4021 to (356, 250, -10) mm, rotated rx -180 ry 0 rz 180 deg; joints [-9.072, -40.734, 102.088, 169.688, 61.745, -175.077]
  MoveL 4022 to (344, 250, -10) mm, rotated rx 180 ry 0 rz 180 deg; joints [-9.141, -41.025, 102.911, 169.661, 62.274, -175.149]
  MoveL 4023 to (343.81, 255.96, -10) mm, rotated rx 180 ry 0 rz -180 deg; joints [-9.356, -41.007, 102.857, 169.415, 62.258, -175.029]
  MoveL 4024 to (343.24, 261.9, -10) mm, rotated rx 180 ry 0 rz -180 deg; joints [-9.573, -40.996, 102.829, 169.17, 62.259, -174.911]
  MoveL 4025 to (342.3, 267.79, -10) mm, rotated rx 180 ry 0 rz 180 deg; joints [-9.79, -40.995, 102.824, 168.926, 62.275, -174.797]
  MoveL 4026 to (340.99, 273.61, -10) mm, rotated rx 180 ry 0 rz 180 deg; joints [-10.006, -41.002, 102.845, 168.683, 62.308, -174.687]
  MoveL 4027 to (339.31, 279.33, -10) mm, rotated rx -180 ry 0 rz -180 deg; joints [-10.222, -41.018, 102.89, 168.444, 62.357, -174.581]
  MoveL 4028 to (337.27, 284.94, -10) mm, rotated rx 180 ry 0 rz -180 deg; joints [-10.436, -41.042, 102.959, 168.208, 62.421, -174.479]
  MoveL 4029 to (334.88, 290.4, -10) mm, rotated rx 180 ry 0 rz 180 deg; joints [-10.648, -41.075, 103.053, 167.977, 62.501, -174.384]
  MoveL 4030 to (332.14, 295.7, -10) mm, rotated rx 180 ry 0 rz -180 deg; joints [-10.857, -41.117, 103.17, 167.751, 62.596, -174.294]
  MoveL 4031 to (329.08, 300.82, -10) mm, rotated rx 180 ry 0 rz -180 deg; joints [-11.061, -41.166, 103.31, 167.532, 62.705, -174.21]
  MoveL 4032 to (325.7, 305.73, -10) mm, rotated rx -180 ry 0 rz -180 deg; joints [-11.262, -41.223, 103.474, 167.32, 62.829, -174.134]
  MoveL 4033 to (322.01, 310.42, -10) mm, rotated rx -180 ry 0 rz -180 deg; joints [-11.457, -41.288, 103.659, 167.115, 62.967, -174.064]
  MoveL 4034 to (318.03, 314.87, -10) mm, rotated rx 180 ry 0 rz -180 deg; joints [-11.646, -41.36, 103.866, 166.92, 63.118, -174.003]
  MoveL 4035 to (313.78, 319.05, -10) mm, rotated rx 180 ry 0 rz 180 deg; joints [-11.828, -41.439, 104.093, 166.734, 63.281, -173.949]
  MoveL 4036 to (309.27, 322.96, -10) mm, rotated rx 180 ry 0 rz -180 deg; joints [-12.003, -41.525, 104.341, 166.557, 63.457, -173.903]
  MoveL 4037 to (304.53, 326.57, -10) mm, rotated rx 180 ry 0 rz -180 deg; joints [-12.17, -41.617, 104.607, 166.392, 63.644, -173.866]
  MoveL 4038 to (299.56, 329.87, -10) mm, rotated rx 180 ry 0 rz -180 deg; joints [-12.329, -41.715, 104.891, 166.238, 63.842, -173.837]
  MoveL 4039 to (294.39, 332.86, -10) mm, rotated rx 180 ry 0 rz -180 deg; joints [-12.478, -41.818, 105.191, 166.096, 64.049, -173.817]
  MoveL 4040 to (289.05, 335.51, -10) mm, rotated rx 180 ry 0 rz 180 deg; joints [-12.618, -41.926, 105.507, 165.966, 64.266, -173.806]
  MoveL 4041 to (283.55, 337.81, -10) mm, rotated rx -180 ry 0 rz -180 deg; joints [-12.747, -42.039, 105.837, 165.849, 64.491, -173.803]
  MoveL 4042 to (277.91, 339.76, -10) mm, rotated rx -180 ry 0 rz 180 deg; joints [-12.865, -42.155, 106.18, 165.745, 64.724, -173.809]
  MoveL 4043 to (272.16, 341.35, -10) mm, rotated rx 180 ry 0 rz 180 deg; joints [-12.972, -42.275, 106.535, 165.655, 64.963, -173.823]
  MoveL 4044 to (266.32, 342.57, -10) mm, rotated rx -180 ry 0 rz -180 deg; joints [-13.067, -42.397, 106.9, 165.58, 65.209, -173.846]
  MoveL 4045 to (260.42, 343.42, -10) mm, rotated rx -180 ry 0 rz -180 deg; joints [-13.149, -42.522, 107.274, 165.519, 65.459, -173.877]
  MoveL 4046 to (254.47, 343.89, -10) mm, rotated rx -180 ry 0 rz 180 deg; joints [-13.218, -42.649, 107.656, 165.472, 65.713, -173.916]
  MoveL 4047 to (248.51, 343.99, -10) mm, rotated rx 180 ry 0 rz 180 deg; joints [-13.273, -42.776, 108.043, 165.441, 65.97, -173.963]
  MoveL 4048 to (242.55, 343.7, -10) mm, rotated rx 180 ry 0 rz 180 deg; joints [-13.315, -42.905, 108.435, 165.424, 66.229, -174.017]
  MoveL 4049 to (236.62, 343.04, -10) mm, rotated rx 180 ry 0 rz 180 deg; joints [-13.343, -43.033, 108.829, 165.423, 66.489, -174.078]
  MoveL 4050 to (230.75, 342.01, -10) mm, rotated rx 180 ry 0 rz 180 deg; joints [-13.356, -43.161, 109.225, 165.438, 66.75, -174.145]
  MoveL 4051 to (224.95, 340.6, -10) mm, rotated rx -180 ry 0 rz 180 deg; joints [-13.355, -43.288, 109.62, 165.468, 67.01, -174.219]
  MoveL 4052 to (219.26, 338.83, -10) mm, rotated rx 180 ry 0 rz -180 deg; joints [-13.339, -43.414, 110.014, 165.513, 67.267, -174.298]
  MoveL 4053 to (213.68, 336.7, -10) mm, rotated rx 180 ry 0 rz 180 deg; joints [-13.309, -43.537, 110.404, 165.574, 67.522, -174.383]
  MoveL 4054 to (208.26, 334.22, -10) mm, rotated rx 180 ry 0 rz -180 deg; joints [-13.263, -43.659, 110.789, 165.65, 67.773, -174.473]
  MoveL 4055 to (203, 331.41, -10) mm, rotated rx -180 ry 0 rz -180 deg; joints [-13.202, -43.777, 111.167, 165.742, 68.019, -174.567]
  MoveL 4056 to (197.93, 328.26, -10) mm, rotated rx -180 ry 0 rz -180 deg; joints [-13.127, -43.892, 111.537, 165.848, 68.26, -174.664]
  MoveL 4057 to (193.07, 324.8, -10) mm, rotated rx 180 ry 0 rz -180 deg; joints [-13.037, -44.003, 111.898, 165.968, 68.493, -174.765]
  MoveL 4058 to (188.44, 321.04, -10) mm, rotated rx 180 ry 0 rz 180 deg; joints [-12.932, -44.11, 112.247, 166.103, 68.719, -174.869]
  MoveL 4059 to (184.06, 316.99, -10) mm, rotated rx -180 ry 0 rz 180 deg; joints [-12.813, -44.212, 112.584, 166.252, 68.936, -174.975]
  MoveL 4060 to (179.95, 312.68, -10) mm, rotated rx 180 ry 0 rz 180 deg; joints [-12.681, -44.309, 112.906, 166.414, 69.144, -175.082]
  MoveL 4061 to (176.11, 308.11, -10) mm, rotated rx 180 ry 0 rz -180 deg; joints [-12.535, -44.401, 113.213, 166.588, 69.341, -175.191]
  MoveL 4062 to (172.57, 303.3, -10) mm, rotated rx 180 ry 0 rz 180 deg; joints [-12.376, -44.488, 113.504, 166.775, 69.526, -175.301]
  MoveL 4063 to (169.35, 298.29, -10) mm, rotated rx -180 ry 0 rz -180 deg; joints [-12.205, -44.568, 113.776, 166.973, 69.699, -175.411]
  MoveL 4064 to (166.45, 293.07, -10) mm, rotated rx 180 ry 0 rz 180 deg; joints [-12.022, -44.643, 114.03, 167.182, 69.859, -175.52]
  MoveL 4065 to (163.89, 287.69, -10) mm, rotated rx 180 ry 0 rz 180 deg; joints [-11.829, -44.711, 114.263, 167.4, 70.005, -175.629]
  MoveL 4066 to (161.67, 282.15, -10) mm, rotated rx 180 ry 0 rz -180 deg; joints [-11.626, -44.773, 114.475, 167.627, 70.136, -175.737]
  MoveL 4067 to (159.81, 276.48, -10) mm, rotated rx -180 ry 0 rz 180 deg; joints [-11.414, -44.828, 114.665, 167.863, 70.253, -175.844]
  MoveL 4068 to (158.31, 270.71, -10) mm, rotated rx -180 ry 0 rz -180 deg; joints [-11.193, -44.876, 114.832, 168.105, 70.353, -175.949]
  MoveL 4069 to (157.18, 264.85, -10) mm, rotated rx -180 ry 0 rz -180 deg; joints [-10.966, -44.917, 114.975, 168.353, 70.437, -176.052]
  MoveL 4070 to (156.43, 258.94, -10) mm, rotated rx -180 ry 0 rz 180 deg; joints [-10.733, -44.951, 115.094, 168.606, 70.504, -176.152]
  MoveL 4071 to (156.05, 252.98, -10) mm, rotated rx -180 ry 0 rz -180 deg; joints [-10.494, -44.978, 115.188, 168.863, 70.554, -176.25]
  MoveL 4072 to (156.05, 247.02, -10) mm, rotated rx 180 ry 0 rz 180 deg; joints [-10.252, -44.997, 115.257, 169.123, 70.587, -176.346]
  MoveL 4073 to (156.43, 241.06, -10) mm, rotated rx -180 ry 0 rz -180 deg; joints [-10.007, -45.01, 115.3, 169.384, 70.602, -176.438]
  MoveL 4074 to (157.18, 235.15, -10) mm, rotated rx 180 ry 0 rz 180 deg; joints [-9.761, -45.015, 115.317, 169.645, 70.599, -176.527]
  MoveL 4075 to (158.31, 229.29, -10) mm, rotated rx -180 ry 0 rz -180 deg; joints [-9.515, -45.012, 115.309, 169.905, 70.578, -176.612]
  MoveL 4076 to (159.81, 223.52, -10) mm, rotated rx -180 ry 0 rz -180 deg; joints [-9.27, -45.003, 115.274, 170.163, 70.54, -176.694]
  MoveL 4077 to (161.67, 217.85, -10) mm, rotated rx 180 ry 0 rz 180 deg; joints [-9.026, -44.985, 115.214, 170.418, 70.484, -176.772]
  MoveL 4078 to (163.89, 212.31, -10) mm, rotated rx 180 ry 0 rz -180 deg; joints [-8.787, -44.961, 115.129, 170.669, 70.41, -176.847]
  MoveL 4079 to (166.45, 206.93, -10) mm, rotated rx -180 ry 0 rz -180 deg; joints [-8.551, -44.93, 115.019, 170.914, 70.32, -176.917]
  MoveL 4080 to (169.35, 201.71, -10) mm, rotated rx 180 ry 0 rz 180 deg; joints [-8.322, -44.891, 114.884, 171.152, 70.213, -176.983]
  MoveL 4081 to (172.57, 196.7, -10) mm, rotated rx -180 ry 0 rz 180 deg; joints [-8.099, -44.845, 114.725, 171.383, 70.089, -177.046]
  MoveL 4082 to (176.11, 191.89, -10) mm, rotated rx -180 ry 0 rz 180 deg; joints [-7.884, -44.793, 114.543, 171.604, 69.95, -177.103]
  MoveL 4083 to (179.95, 187.32, -10) mm, rotated rx -180 ry 0 rz 180 deg; joints [-7.677, -44.733, 114.339, 171.816, 69.796, -177.157]
  MoveL 4084 to (184.06, 183.01, -10) mm, rotated rx -180 ry 0 rz -180 deg; joints [-7.48, -44.667, 114.113, 172.017, 69.628, -177.205]
  MoveL 4085 to (188.44, 178.96, -10) mm, rotated rx 180 ry 0 rz 180 deg; joints [-7.294, -44.595, 113.866, 172.207, 69.447, -177.249]
  MoveL 4086 to (193.07, 175.2, -10) mm, rotated rx 180 ry 0 rz 180 deg; joints [-7.119, -44.516, 113.6, 172.384, 69.252, -177.288]
  MoveL 4087 to (197.93, 171.74, -10) mm, rotated rx 180 ry 0 rz 180 deg; joints [-6.956, -44.432, 113.316, 172.549, 69.047, -177.322]
  MoveL 4088 to (203, 168.59, -10) mm, rotated rx -180 ry 0 rz 180 deg; joints [-6.806, -44.342, 113.014, 172.699, 68.83, -177.351]
  MoveL 4089 to (208.26, 165.78, -10) mm, rotated rx -180 ry 0 rz 180 deg; joints [-6.668, -44.246, 112.697, 172.836, 68.604, -177.374]
  MoveL 4090 to (213.68, 163.3, -10) mm, rotated rx -180 ry 0 rz -180 deg; joints [-6.545, -44.146, 112.365, 172.957, 68.368, -177.392]
  MoveL 4091 to (219.26, 161.17, -10) mm, rotated rx -180 ry 0 rz -180 deg; joints [-6.435, -44.04, 112.02, 173.063, 68.125, -177.405]
  MoveL 4092 to (224.95, 159.4, -10) mm, rotated rx 180 ry 0 rz -180 deg; joints [-6.34, -43.931, 111.663, 173.154, 67.876, -177.411]
  MoveL 4093 to (230.75, 157.99, -10) mm, rotated rx -180 ry 0 rz -180 deg; joints [-6.259, -43.817, 111.296, 173.229, 67.621, -177.412]
  MoveL 4094 to (236.62, 156.96, -10) mm, rotated rx 180 ry 0 rz 180 deg; joints [-6.194, -43.7, 110.92, 173.287, 67.361, -177.406]
  MoveL 4095 to (242.55, 156.3, -10) mm, rotated rx 180 ry 0 rz 180 deg; joints [-6.143, -43.58, 110.537, 173.329, 67.098, -177.394]
  MoveL 4096 to (248.51, 156.01, -10) mm, rotated rx -180 ry 0 rz -180 deg; joints [-6.107, -43.457, 110.149, 173.355, 66.832, -177.376]
  MoveL 4097 to (254.47, 156.11, -10) mm, rotated rx -180 ry 0 rz -180 deg; joints [-6.086, -43.332, 109.757, 173.365, 66.566, -177.351]
  MoveL 4098 to (260.42, 156.58, -10) mm, rotated rx -180 ry 0 rz -180 deg; joints [-6.08, -43.205, 109.362, 173.358, 66.299, -177.32]
  MoveL 4099 to (266.32, 157.43, -10) mm, rotated rx -180 ry 0 rz -180 deg; joints [-6.088, -43.077, 108.966, 173.335, 66.033, -177.282]
  MoveL 4100 to (272.16, 158.65, -10) mm, rotated rx 180 ry 0 rz -180 deg; joints [-6.111, -42.949, 108.571, 173.296, 65.769, -177.238]
  MoveL 4101 to (277.91, 160.24, -10) mm, rotated rx 180 ry 0 rz 180 deg; joints [-6.148, -42.821, 108.178, 173.241, 65.508, -177.187]
  MoveL 4102 to (283.55, 162.19, -10) mm, rotated rx 180 ry 0 rz 180 deg; joints [-6.199, -42.693, 107.789, 173.171, 65.252, -177.13]
  MoveL 4103 to (289.05, 164.49, -10) mm, rotated rx -180 ry 0 rz -180 deg; joints [-6.263, -42.566, 107.405, 173.086, 65, -177.066]
  MoveL 4104 to (294.39, 167.14, -10) mm, rotated rx 180 ry 0 rz 180 deg; joints [-6.341, -42.44, 107.029, 172.986, 64.755, -176.996]
  MoveL 4105 to (299.56, 170.13, -10) mm, rotated rx 180 ry 0 rz 180 deg; joints [-6.431, -42.317, 106.66, 172.872, 64.517, -176.92]
  MoveL 4106 to (304.53, 173.43, -10) mm, rotated rx 180 ry 0 rz 180 deg; joints [-6.534, -42.196, 106.302, 172.744, 64.286, -176.838]
  MoveL 4107 to (309.27, 177.04, -10) mm, rotated rx 180 ry 0 rz -180 deg; joints [-6.648, -42.079, 105.954, 172.603, 64.065, -176.75]
  MoveL 4108 to (313.78, 180.95, -10) mm, rotated rx 180 ry 0 rz 180 deg; joints [-6.773, -41.965, 105.619, 172.45, 63.853, -176.657]
  MoveL 4109 to (318.03, 185.13, -10) mm, rotated rx -180 ry 0 rz -180 deg; joints [-6.909, -41.855, 105.298, 172.285, 63.651, -176.559]
  MoveL 4110 to (322.01, 189.58, -10) mm, rotated rx -180 ry 0 rz 180 deg; joints [-7.056, -41.75, 104.992, 172.108, 63.461, -176.456]
  MoveL 4111 to (325.7, 194.27, -10) mm, rotated rx -180 ry 0 rz -180 deg; joints [-7.211, -41.65, 104.703, 171.922, 63.282, -176.349]
  MoveL 4112 to (329.08, 199.18, -10) mm, rotated rx -180 ry 0 rz 180 deg; joints [-7.375, -41.556, 104.43, 171.725, 63.117, -176.237]
  MoveL 4113 to (332.14, 204.3, -10) mm, rotated rx -180 ry 0 rz -180 deg; joints [-7.548, -41.468, 104.177, 171.52, 62.964, -176.123]
  MoveL 4114 to (334.88, 209.6, -10) mm, rotated rx 180 ry 0 rz 180 deg; joints [-7.728, -41.387, 103.942, 171.306, 62.825, -176.005]
  MoveL 4115 to (337.27, 215.06, -10) mm, rotated rx 180 ry 0 rz 180 deg; joints [-7.915, -41.312, 103.728, 171.086, 62.701, -175.885]
  MoveL 4116 to (339.31, 220.67, -10) mm, rotated rx 180 ry 0 rz -180 deg; joints [-8.108, -41.245, 103.535, 170.859, 62.591, -175.764]
  MoveL 4117 to (340.99, 226.39, -10) mm, rotated rx 180 ry 0 rz 180 deg; joints [-8.306, -41.185, 103.364, 170.626, 62.496, -175.641]
  MoveL 4118 to (342.3, 232.21, -10) mm, rotated rx 180 ry 0 rz -180 deg; joints [-8.509, -41.133, 103.216, 170.39, 62.417, -175.517]
  MoveL 4119 to (343.24, 238.1, -10) mm, rotated rx -180 ry 0 rz -180 deg; joints [-8.717, -41.089, 103.09, 170.149, 62.353, -175.393]
  MoveL 4120 to (343.81, 244.04, -10) mm, rotated rx 180 ry 0 rz -180 deg; joints [-8.928, -41.053, 102.989, 169.906, 62.305, -175.27]
  MoveL 4121 to (344, 250, -10) mm, rotated rx 180 ry 0 rz 180 deg; joints [-9.141, -41.025, 102.911, 169.661, 62.274, -175.149]
  MoveL 4122 to (332, 250, -10) mm, rotated rx -180 ry 0 rz 180 deg; joints [-9.211, -41.312, 103.729, 169.632, 62.801, -175.22]
  MoveL 4123 to (331.83, 255.2, -10) mm, rotated rx -180 ry 0 rz -180 deg; joints [-9.4, -41.296, 103.682, 169.417, 62.788, -175.117]
  MoveL 4124 to (331.34, 260.38, -10) mm, rotated rx -180 ry 0 rz 180 deg; joints [-9.59, -41.287, 103.657, 169.203, 62.788, -175.016]
  MoveL 4125 to (330.52, 265.52, -10) mm, rotated rx 180 ry 0 rz 180 deg; joints [-9.781, -41.286, 103.653, 168.989, 62.802, -174.918]
  MoveL 4126 to (329.37, 270.59, -10) mm, rotated rx 180 ry 0 rz -180 deg; joints [-9.972, -41.292, 103.671, 168.776, 62.831, -174.823]
  MoveL 4127 to (327.91, 275.59, -10) mm, rotated rx 180 ry 0 rz -180 deg; joints [-10.161, -41.306, 103.71, 168.567, 62.873, -174.731]
  MoveL 4128 to (326.13, 280.48, -10) mm, rotated rx 180 ry 0 rz 180 deg; joints [-10.349, -41.327, 103.771, 168.36, 62.929, -174.644]
  MoveL 4129 to (324.04, 285.24, -10) mm, rotated rx 180 ry 0 rz 180 deg; joints [-10.535, -41.356, 103.852, 168.158, 62.999, -174.562]
  MoveL 4130 to (321.66, 289.87, -10) mm, rotated rx -180 ry 0 rz -180 deg; joints [-10.719, -41.391, 103.955, 167.96, 63.081, -174.485]
  MoveL 4131 to (318.98, 294.33, -10) mm, rotated rx -180 ry 0 rz -180 deg; joints [-10.898, -41.434, 104.078, 167.768, 63.177, -174.413]
  MoveL 4132 to (316.03, 298.62, -10) mm, rotated rx -180 ry 0 rz 180 deg; joints [-11.074, -41.484, 104.22, 167.583, 63.285, -174.347]
  MoveL 4133 to (312.82, 302.71, -10) mm, rotated rx 180 ry 0 rz -180 deg; joints [-11.245, -41.54, 104.382, 167.404, 63.406, -174.287]
  MoveL 4134 to (309.35, 306.59, -10) mm, rotated rx 180 ry 0 rz 180 deg; joints [-11.411, -41.602, 104.563, 167.233, 63.537, -174.234]
  MoveL 4135 to (305.64, 310.24, -10) mm, rotated rx -180 ry 0 rz 180 deg; joints [-11.57, -41.671, 104.762, 167.07, 63.681, -174.188]
  MoveL 4136 to (301.71, 313.64, -10) mm, rotated rx -180 ry 0 rz -180 deg; joints [-11.724, -41.745, 104.978, 166.915, 63.834, -174.148]
  MoveL 4137 to (297.56, 316.8, -10) mm, rotated rx -180 ry 0 rz -180 deg; joints [-11.87, -41.825, 105.211, 166.771, 63.998, -174.116]
  MoveL 4138 to (293.23, 319.68, -10) mm, rotated rx 180 ry 0 rz -180 deg; joints [-12.008, -41.91, 105.459, 166.636, 64.171, -174.09]
  MoveL 4139 to (288.73, 322.28, -10) mm, rotated rx -180 ry 0 rz 180 deg; joints [-12.138, -41.999, 105.721, 166.511, 64.353, -174.073]
  MoveL 4140 to (284.06, 324.59, -10) mm, rotated rx -180 ry 0 rz 180 deg; joints [-12.26, -42.093, 105.997, 166.398, 64.542, -174.062]
  MoveL 4141 to (279.26, 326.6, -10) mm, rotated rx 180 ry 0 rz -180 deg; joints [-12.372, -42.191, 106.286, 166.296, 64.739, -174.059]
  MoveL 4142 to (274.35, 328.3, -10) mm, rotated rx 180 ry 0 rz -180 deg; joints [-12.474, -42.292, 106.585, 166.206, 64.943, -174.064]
  MoveL 4143 to (269.33, 329.69, -10) mm, rotated rx 180 ry 0 rz -180 deg; joints [-12.566, -42.396, 106.895, 166.127, 65.153, -174.075]
  MoveL 4144 to (264.24, 330.75, -10) mm, rotated rx -180 ry 0 rz 180 deg; joints [-12.648, -42.502, 107.214, 166.062, 65.367, -174.094]
  MoveL 4145 to (259.09, 331.49, -10) mm, rotated rx 180 ry 0 rz -180 deg; joints [-12.718, -42.61, 107.541, 166.009, 65.586, -174.12]
  MoveL 4146 to (253.9, 331.91, -10) mm, rotated rx 180 ry 0 rz -180 deg; joints [-12.777, -42.72, 107.874, 165.969, 65.808, -174.153]
  MoveL 4147 to (248.7, 331.99, -10) mm, rotated rx 180 ry 0 rz 180 deg; joints [-12.824, -42.832, 108.212, 165.942, 66.033, -174.192]
  MoveL 4148 to (243.5, 331.74, -10) mm, rotated rx 180 ry 0 rz 180 deg; joints [-12.859, -42.943, 108.554, 165.929, 66.26, -174.238]
  MoveL 4149 to (238.33, 331.17, -10) mm, rotated rx -180 ry 0 rz -180 deg; joints [-12.882, -43.055, 108.898, 165.929, 66.488, -174.29]
  MoveL 4150 to (233.21, 330.26, -10) mm, rotated rx 180 ry 0 rz -180 deg; joints [-12.892, -43.167, 109.243, 165.942, 66.715, -174.347]
  MoveL 4151 to (228.15, 329.04, -10) mm, rotated rx 180 ry 0 rz 180 deg; joints [-12.89, -43.278, 109.588, 165.969, 66.942, -174.41]
  MoveL 4152 to (223.18, 327.49, -10) mm, rotated rx -180 ry 0 rz 180 deg; joints [-12.874, -43.388, 109.931, 166.01, 67.167, -174.478]
  MoveL 4153 to (218.32, 325.63, -10) mm, rotated rx -180 ry 0 rz -180 deg; joints [-12.846, -43.496, 110.271, 166.064, 67.39, -174.55]
  MoveL 4154 to (213.59, 323.47, -10) mm, rotated rx 180 ry 0 rz -180 deg; joints [-12.804, -43.602, 110.607, 166.132, 67.609, -174.627]
  MoveL 4155 to (209, 321.01, -10) mm, rotated rx 180 ry 0 rz -180 deg; joints [-12.75, -43.705, 110.937, 166.212, 67.823, -174.708]
  MoveL 4156 to (204.58, 318.27, -10) mm, rotated rx -180 ry 0 rz -180 deg; joints [-12.683, -43.806, 111.259, 166.306, 68.033, -174.792]
  MoveL 4157 to (200.34, 315.25, -10) mm, rotated rx 180 ry 0 rz -180 deg; joints [-12.603, -43.903, 111.573, 166.412, 68.236, -174.879]
  MoveL 4158 to (196.3, 311.97, -10) mm, rotated rx -180 ry 0 rz 180 deg; joints [-12.51, -43.997, 111.877, 166.531, 68.433, -174.968]
  MoveL 4159 to (192.48, 308.44, -10) mm, rotated rx 180 ry 0 rz 180 deg; joints [-12.406, -44.086, 112.171, 166.661, 68.621, -175.06]
  MoveL 4160 to (188.89, 304.68, -10) mm, rotated rx 180 ry 0 rz 180 deg; joints [-12.29, -44.172, 112.451, 166.803, 68.802, -175.153]
  MoveL 4161 to (185.54, 300.69, -10) mm, rotated rx -180 ry 0 rz 180 deg; joints [-12.162, -44.253, 112.719, 166.956, 68.972, -175.248]
  MoveL 4162 to (182.46, 296.5, -10) mm, rotated rx 180 ry 0 rz -180 deg; joints [-12.023, -44.329, 112.971, 167.119, 69.133, -175.343]
  MoveL 4163 to (179.65, 292.12, -10) mm, rotated rx 180 ry 0 rz 180 deg; joints [-11.874, -44.4, 113.209, 167.292, 69.283, -175.439]
  MoveL 4164 to (177.12, 287.57, -10) mm, rotated rx 180 ry 0 rz 180 deg; joints [-11.715, -44.466, 113.429, 167.474, 69.422, -175.535]
  MoveL 4165 to (174.88, 282.88, -10) mm, rotated rx 180 ry 0 rz -180 deg; joints [-11.547, -44.526, 113.632, 167.664, 69.548, -175.63]
  MoveL 4166 to (172.95, 278.05, -10) mm, rotated rx 180 ry 0 rz 180 deg; joints [-11.37, -44.58, 113.816, 167.863, 69.662, -175.725]
  MoveL 4167 to (171.32, 273.1, -10) mm, rotated rx -180 ry 0 rz 180 deg; joints [-11.186, -44.629, 113.981, 168.067, 69.762, -175.819]
  MoveL 4168 to (170.01, 268.07, -10) mm, rotated rx -180 ry 0 rz 180 deg; joints [-10.995, -44.671, 114.126, 168.278, 69.849, -175.911]
  MoveL 4169 to (169.03, 262.96, -10) mm, rotated rx -180 ry 0 rz -180 deg; joints [-10.798, -44.708, 114.251, 168.494, 69.921, -176.002]
  MoveL 4170 to (168.37, 257.79, -10) mm, rotated rx 180 ry 0 rz -180 deg; joints [-10.596, -44.738, 114.354, 168.714, 69.979, -176.091]
  MoveL 4171 to (168.04, 252.6, -10) mm, rotated rx -180 ry 0 rz 180 deg; joints [-10.389, -44.761, 114.436, 168.937, 70.022, -176.178]
  MoveL 4172 to (168.04, 247.4, -10) mm, rotated rx -180 ry 0 rz -180 deg; joints [-10.18, -44.779, 114.495, 169.162, 70.05, -176.263]
  MoveL 4173 to (168.37, 242.21, -10) mm, rotated rx -180 ry 0 rz 180 deg; joints [-9.968, -44.79, 114.533, 169.389, 70.062, -176.345]
  MoveL 4174 to (169.03, 237.04, -10) mm, rotated rx 180 ry 0 rz 180 deg; joints [-9.755, -44.794, 114.548, 169.616, 70.059, -176.424]
  MoveL 4175 to (170.01, 231.93, -10) mm, rotated rx 180 ry 0 rz -180 deg; joints [-9.542, -44.792, 114.541, 169.842, 70.041, -176.5]
  MoveL 4176 to (171.32, 226.9, -10) mm, rotated rx 180 ry 0 rz -180 deg; joints [-9.33, -44.783, 114.511, 170.066, 70.007, -176.573]
  MoveL 4177 to (172.95, 221.95, -10) mm, rotated rx 180 ry 0 rz 180 deg; joints [-9.12, -44.768, 114.459, 170.287, 69.958, -176.643]
  MoveL 4178 to (174.88, 217.12, -10) mm, rotated rx 180 ry 0 rz 180 deg; joints [-8.912, -44.747, 114.385, 170.504, 69.895, -176.709]
  MoveL 4179 to (177.12, 212.43, -10) mm, rotated rx -180 ry 0 rz -180 deg; joints [-8.709, -44.719, 114.289, 170.717, 69.816, -176.772]
  MoveL 4180 to (179.65, 207.88, -10) mm, rotated rx 180 ry 0 rz 180 deg; joints [-8.51, -44.684, 114.172, 170.924, 69.723, -176.831]
  MoveL 4181 to (182.46, 203.5, -10) mm, rotated rx 180 ry 0 rz 180 deg; joints [-8.316, -44.644, 114.034, 171.124, 69.616, -176.886]
  MoveL 4182 to (185.54, 199.31, -10) mm, rotated rx 180 ry 0 rz 180 deg; joints [-8.13, -44.598, 113.875, 171.316, 69.495, -176.938]
  MoveL 4183 to (188.89, 195.32, -10) mm, rotated rx 180 ry 0 rz 180 deg; joints [-7.95, -44.545, 113.698, 171.5, 69.362, -176.985]
  MoveL 4184 to (192.48, 191.56, -10) mm, rotated rx 180 ry 0 rz -180 deg; joints [-7.779, -44.487, 113.501, 171.675, 69.216, -177.028]
  MoveL 4185 to (196.3, 188.03, -10) mm, rotated rx 180 ry 0 rz -180 deg; joints [-7.617, -44.423, 113.287, 171.841, 69.059, -177.066]
  MoveL 4186 to (200.34, 184.75, -10) mm, rotated rx 180 ry 0 rz 180 deg; joints [-7.465, -44.354, 113.055, 171.995, 68.89, -177.101]
  MoveL 4187 to (204.58, 181.73, -10) mm, rotated rx 180 ry 0 rz -180 deg; joints [-7.322, -44.28, 112.808, 172.138, 68.712, -177.13]
  MoveL 4188 to (209, 178.99, -10) mm, rotated rx -180 ry 0 rz 180 deg; joints [-7.191, -44.2, 112.545, 172.27, 68.524, -177.155]
  MoveL 4189 to (213.59, 176.53, -10) mm, rotated rx 180 ry 0 rz 180 deg; joints [-7.07, -44.116, 112.269, 172.389, 68.327, -177.175]
  MoveL 4190 to (218.32, 174.37, -10) mm, rotated rx 180 ry 0 rz 180 deg; joints [-6.962, -44.028, 111.98, 172.495, 68.123, -177.19]
  MoveL 4191 to (223.18, 172.51, -10) mm, rotated rx 180 ry 0 rz 180 deg; joints [-6.865, -43.936, 111.679, 172.588, 67.912, -177.2]
  MoveL 4192 to (228.15, 170.96, -10) mm, rotated rx -180 ry 0 rz -180 deg; joints [-6.781, -43.84, 111.369, 172.668, 67.695, -177.204]
  MoveL 4193 to (233.21, 169.74, -10) mm, rotated rx 180 ry 0 rz 180 deg; joints [-6.709, -43.74, 111.049, 172.734, 67.473, -177.203]
  MoveL 4194 to (238.33, 168.83, -10) mm, rotated rx 180 ry 0 rz -180 deg; joints [-6.65, -43.638, 110.721, 172.785, 67.247, -177.197]
  MoveL 4195 to (243.5, 168.26, -10) mm, rotated rx -180 ry 0 rz 180 deg; joints [-6.605, -43.532, 110.388, 172.823, 67.018, -177.185]
  MoveL 4196 to (248.7, 168.01, -10) mm, rotated rx 180 ry 0 rz -180 deg; joints [-6.572, -43.425, 110.049, 172.847, 66.787, -177.168]
  MoveL 4197 to (253.9, 168.09, -10) mm, rotated rx 180 ry 0 rz -180 deg; joints [-6.552, -43.316, 109.707, 172.856, 66.554, -177.145]
  MoveL 4198 to (259.09, 168.51, -10) mm, rotated rx 180 ry 0 rz -180 deg; joints [-6.545, -43.205, 109.362, 172.851, 66.322, -177.116]
  MoveL 4199 to (264.24, 169.25, -10) mm, rotated rx -180 ry 0 rz -180 deg; joints [-6.55, -43.094, 109.017, 172.832, 66.09, -177.082]
  MoveL 4200 to (269.33, 170.31, -10) mm, rotated rx 180 ry 0 rz 180 deg; joints [-6.569, -42.982, 108.672, 172.799, 65.86, -177.042]
  MoveL 4201 to (274.35, 171.7, -10) mm, rotated rx 180 ry 0 rz 180 deg; joints [-6.6, -42.87, 108.329, 172.752, 65.633, -176.996]
  MoveL 4202 to (279.26, 173.4, -10) mm, rotated rx 180 ry 0 rz -180 deg; joints [-6.643, -42.759, 107.99, 172.691, 65.409, -176.945]
  MoveL 4203 to (284.06, 175.41, -10) mm, rotated rx -180 ry 0 rz 180 deg; joints [-6.697, -42.648, 107.655, 172.618, 65.189, -176.888]
  MoveL 4204 to (288.73, 177.72, -10) mm, rotated rx -180 ry 0 rz 180 deg; joints [-6.764, -42.539, 107.326, 172.531, 64.975, -176.826]
  MoveL 4205 to (293.23, 180.32, -10) mm, rotated rx 180 ry 0 rz -180 deg; joints [-6.842, -42.432, 107.004, 172.433, 64.766, -176.758]
  MoveL 4206 to (297.56, 183.2, -10) mm, rotated rx 180 ry 0 rz 180 deg; joints [-6.93, -42.327, 106.691, 172.322, 64.565, -176.686]
  MoveL 4207 to (301.71, 186.36, -10) mm, rotated rx 180 ry 0 rz -180 deg; joints [-7.029, -42.225, 106.388, 172.199, 64.371, -176.609]
  MoveL 4208 to (305.64, 189.76, -10) mm, rotated rx 180 ry 0 rz 180 deg; joints [-7.138, -42.126, 106.095, 172.066, 64.186, -176.527]
  MoveL 4209 to (309.35, 193.41, -10) mm, rotated rx -180 ry 0 rz 180 deg; joints [-7.256, -42.031, 105.815, 171.922, 64.009, -176.441]
  MoveL 4210 to (312.82, 197.29, -10) mm, rotated rx -180 ry 0 rz -180 deg; joints [-7.383, -41.94, 105.548, 171.769, 63.843, -176.351]
  MoveL 4211 to (316.03, 201.38, -10) mm, rotated rx 180 ry 0 rz 180 deg; joints [-7.519, -41.854, 105.294, 171.606, 63.687, -176.258]
  MoveL 4212 to (318.98, 205.67, -10) mm, rotated rx -180 ry 0 rz -180 deg; joints [-7.663, -41.772, 105.057, 171.435, 63.542, -176.161]
  MoveL 4213 to (321.66, 210.13, -10) mm, rotated rx -180 ry 0 rz 180 deg; joints [-7.813, -41.696, 104.835, 171.256, 63.408, -176.061]
  MoveL 4214 to (324.04, 214.76, -10) mm, rotated rx -180 ry 0 rz 180 deg; joints [-7.971, -41.625, 104.63, 171.069, 63.286, -175.959]
  MoveL 4215 to (326.13, 219.52, -10) mm, rotated rx 180 ry 0 rz -180 deg; joints [-8.134, -41.561, 104.443, 170.877, 63.177, -175.855]
  MoveL 4216 to (327.91, 224.41, -10) mm, rotated rx -180 ry 0 rz 180 deg; joints [-8.304, -41.502, 104.274, 170.679, 63.081, -175.75]
  MoveL 4217 to (329.37, 229.41, -10) mm, rotated rx -180 ry 0 rz 180 deg; joints [-8.478, -41.45, 104.125, 170.476, 62.997, -175.644]
  MoveL 4218 to (330.52, 234.48, -10) mm, rotated rx -180 ry 0 rz -180 deg; joints [-8.656, -41.405, 103.995, 170.269, 62.928, -175.537]
  MoveL 4219 to (331.34, 239.62, -10) mm, rotated rx -180 ry 0 rz 180 deg; joints [-8.838, -41.367, 103.885, 170.059, 62.872, -175.431]
  MoveL 4220 to (331.83, 244.8, -10) mm, rotated rx -180 ry 0 rz -180 deg; joints [-9.023, -41.336, 103.796, 169.846, 62.83, -175.325]
  MoveL 4221 to (332, 250, -10) mm, rotated rx -180 ry 0 rz 180 deg; joints [-9.211, -41.312, 103.729, 169.632, 62.801, -175.22]
  MoveL 4222 to (320, 250, -10) mm, rotated rx -180 ry 0 rz -180 deg; joints [-9.282, -41.595, 104.541, 169.601, 63.329, -175.291]
  MoveL 4223 to (319.86, 254.44, -10) mm, rotated rx -180 ry 0 rz 180 deg; joints [-9.445, -41.581, 104.502, 169.417, 63.317, -175.204]
  MoveL 4224 to (319.44, 258.86, -10) mm, rotated rx 180 ry 0 rz -180 deg; joints [-9.608, -41.573, 104.48, 169.234, 63.317, -175.119]
  MoveL 4225 to (318.74, 263.25, -10) mm, rotated rx 180 ry 0 rz -180 deg; joints [-9.772, -41.572, 104.477, 169.05, 63.329, -175.037]
  MoveL 4226 to (317.76, 267.58, -10) mm, rotated rx -180 ry 0 rz -180 deg; joints [-9.936, -41.578, 104.492, 168.869, 63.353, -174.957]
  MoveL 4227 to (316.5, 271.84, -10) mm, rotated rx 180 ry 0 rz -180 deg; joints [-10.099, -41.589, 104.526, 168.689, 63.389, -174.88]
  MoveL 4228 to (314.99, 276.02, -10) mm, rotated rx 180 ry 0 rz 180 deg; joints [-10.261, -41.607, 104.577, 168.512, 63.437, -174.807]
  MoveL 4229 to (313.2, 280.09, -10) mm, rotated rx -180 ry 0 rz 180 deg; joints [-10.421, -41.631, 104.647, 168.339, 63.496, -174.738]
  MoveL 4230 to (311.17, 284.03, -10) mm, rotated rx 180 ry 0 rz 180 deg; joints [-10.579, -41.662, 104.735, 168.17, 63.567, -174.673]
  MoveL 4231 to (308.89, 287.84, -10) mm, rotated rx 180 ry 0 rz 180 deg; joints [-10.733, -41.698, 104.84, 168.005, 63.649, -174.612]
  MoveL 4232 to (306.37, 291.5, -10) mm, rotated rx -180 ry 0 rz -180 deg; joints [-10.884, -41.74, 104.962, 167.846, 63.741, -174.557]
  MoveL 4233 to (303.62, 295, -10) mm, rotated rx 180 ry 0 rz 180 deg; joints [-11.03, -41.787, 105.101, 167.692, 63.844, -174.507]
  MoveL 4234 to (300.66, 298.31, -10) mm, rotated rx 180 ry 0 rz -180 deg; joints [-11.172, -41.84, 105.255, 167.546, 63.957, -174.462]
  MoveL 4235 to (297.5, 301.42, -10) mm, rotated rx 180 ry 0 rz -180 deg; joints [-11.309, -41.899, 105.425, 167.406, 64.08, -174.422]
  MoveL 4236 to (294.14, 304.33, -10) mm, rotated rx 180 ry 0 rz -180 deg; joints [-11.44, -41.962, 105.61, 167.274, 64.211, -174.389]
  MoveL 4237 to (290.6, 307.02, -10) mm, rotated rx -180 ry 0 rz 180 deg; joints [-11.565, -42.029, 105.809, 167.15, 64.351, -174.361]
  MoveL 4238 to (286.91, 309.48, -10) mm, rotated rx 180 ry 0 rz 180 deg; joints [-11.683, -42.101, 106.021, 167.035, 64.5, -174.339]
  MoveL 4239 to (283.06, 311.7, -10) mm, rotated rx 180 ry 0 rz 180 deg; joints [-11.794, -42.177, 106.246, 166.928, 64.655, -174.324]
  MoveL 4240 to (279.08, 313.67, -10) mm, rotated rx -180 ry 0 rz 180 deg; joints [-11.898, -42.257, 106.482, 166.831, 64.818, -174.315]
  MoveL 4241 to (274.98, 315.39, -10) mm, rotated rx 180 ry 0 rz 180 deg; joints [-11.993, -42.34, 106.728, 166.744, 64.987, -174.312]
  MoveL 4242 to (270.78, 316.84, -10) mm, rotated rx -180 ry 0 rz -180 deg; joints [-12.08, -42.425, 106.984, 166.667, 65.161, -174.315]
  MoveL 4243 to (266.5, 318.03, -10) mm, rotated rx -180 ry 0 rz -180 deg; joints [-12.158, -42.514, 107.249, 166.601, 65.341, -174.324]
  MoveL 4244 to (262.16, 318.94, -10) mm, rotated rx 180 ry 0 rz -180 deg; joints [-12.226, -42.604, 107.522, 166.545, 65.524, -174.339]
  MoveL 4245 to (257.76, 319.57, -10) mm, rotated rx -180 ry 0 rz -180 deg; joints [-12.285, -42.696, 107.801, 166.5, 65.712, -174.36]
  MoveL 4246 to (253.33, 319.92, -10) mm, rotated rx 180 ry 0 rz 180 deg; joints [-12.335, -42.79, 108.085, 166.466, 65.902, -174.387]
  MoveL 4247 to (248.89, 319.99, -10) mm, rotated rx 180 ry 0 rz -180 deg; joints [-12.374, -42.885, 108.374, 166.444, 66.095, -174.42]
  MoveL 4248 to (244.45, 319.78, -10) mm, rotated rx 180 ry 0 rz 180 deg; joints [-12.402, -42.98, 108.666, 166.433, 66.289, -174.457]
  MoveL 4249 to (240.04, 319.29, -10) mm, rotated rx -180 ry 0 rz 180 deg; joints [-12.42, -43.076, 108.96, 166.434, 66.483, -174.5]
  MoveL 4250 to (235.66, 318.52, -10) mm, rotated rx 180 ry 0 rz -180 deg; joints [-12.428, -43.171, 109.255, 166.446, 66.678, -174.548]
  MoveL 4251 to (231.35, 317.47, -10) mm, rotated rx 180 ry 0 rz 180 deg; joints [-12.424, -43.265, 109.549, 166.47, 66.872, -174.601]
  MoveL 4252 to (227.11, 316.15, -10) mm, rotated rx 180 ry 0 rz -180 deg; joints [-12.409, -43.359, 109.842, 166.506, 67.064, -174.658]
  MoveL 4253 to (222.96, 314.56, -10) mm, rotated rx -180 ry 0 rz -180 deg; joints [-12.384, -43.451, 110.132, 166.553, 67.254, -174.718]
  MoveL 4254 to (218.92, 312.72, -10) mm, rotated rx -180 ry 0 rz 180 deg; joints [-12.347, -43.542, 110.419, 166.612, 67.441, -174.783]
  MoveL 4255 to (215, 310.62, -10) mm, rotated rx -180 ry 0 rz -180 deg; joints [-12.299, -43.631, 110.7, 166.681, 67.624, -174.85]
  MoveL 4256 to (211.23, 308.28, -10) mm, rotated rx 180 ry 0 rz -180 deg; joints [-12.241, -43.717, 110.975, 166.762, 67.803, -174.921]
  MoveL 4257 to (207.61, 305.7, -10) mm, rotated rx -180 ry 0 rz 180 deg; joints [-12.172, -43.8, 111.243, 166.854, 67.976, -174.995]
  MoveL 4258 to (204.16, 302.9, -10) mm, rotated rx 180 ry 0 rz -180 deg; joints [-12.092, -43.881, 111.502, 166.955, 68.143, -175.07]
  MoveL 4259 to (200.9, 299.89, -10) mm, rotated rx -180 ry 0 rz -180 deg; joints [-12.002, -43.958, 111.752, 167.067, 68.304, -175.148]
  MoveL 4260 to (197.83, 296.67, -10) mm, rotated rx -180 ry 0 rz 180 deg; joints [-11.902, -44.031, 111.991, 167.189, 68.457, -175.227]
  MoveL 4261 to (194.98, 293.27, -10) mm, rotated rx -180 ry 0 rz -180 deg; joints [-11.793, -44.101, 112.219, 167.32, 68.602, -175.307]
  MoveL 4262 to (192.34, 289.69, -10) mm, rotated rx -180 ry 0 rz -180 deg; joints [-11.674, -44.167, 112.434, 167.46, 68.739, -175.389]
  MoveL 4263 to (189.94, 285.96, -10) mm, rotated rx -180 ry 0 rz -180 deg; joints [-11.547, -44.228, 112.636, 167.608, 68.866, -175.47]
  MoveL 4264 to (187.78, 282.08, -10) mm, rotated rx -180 ry 0 rz -180 deg; joints [-11.412, -44.284, 112.823, 167.763, 68.984, -175.552]
  MoveL 4265 to (185.87, 278.07, -10) mm, rotated rx -180 ry 0 rz 180 deg; joints [-11.269, -44.336, 112.996, 167.926, 69.091, -175.634]
  MoveL 4266 to (184.22, 273.94, -10) mm, rotated rx 180 ry 0 rz 180 deg; joints [-11.118, -44.383, 113.153, 168.094, 69.187, -175.716]
  MoveL 4267 to (182.84, 269.72, -10) mm, rotated rx -180 ry 0 rz -180 deg; joints [-10.962, -44.425, 113.293, 168.269, 69.272, -175.796]
  MoveL 4268 to (181.72, 265.42, -10) mm, rotated rx 180 ry 0 rz -180 deg; joints [-10.8, -44.462, 113.417, 168.448, 69.345, -175.876]
  MoveL 4269 to (180.88, 261.06, -10) mm, rotated rx -180 ry 0 rz 180 deg; joints [-10.633, -44.493, 113.522, 168.632, 69.406, -175.955]
  MoveL 4270 to (180.32, 256.65, -10) mm, rotated rx -180 ry 0 rz -180 deg; joints [-10.461, -44.519, 113.61, 168.819, 69.454, -176.032]
  MoveL 4271 to (180.04, 252.22, -10) mm, rotated rx 180 ry 0 rz 180 deg; joints [-10.287, -44.54, 113.68, 169.009, 69.49, -176.107]
  MoveL 4272 to (180.04, 247.78, -10) mm, rotated rx -180 ry 0 rz 180 deg; joints [-10.109, -44.555, 113.731, 169.2, 69.514, -176.181]
  MoveL 4273 to (180.32, 243.35, -10) mm, rotated rx -180 ry 0 rz -180 deg; joints [-9.93, -44.564, 113.762, 169.393, 69.524, -176.252]
  MoveL 4274 to (180.88, 238.94, -10) mm, rotated rx 180 ry 0 rz 180 deg; joints [-9.75, -44.568, 113.775, 169.585, 69.521, -176.321]
  MoveL 4275 to (181.72, 234.58, -10) mm, rotated rx -180 ry 0 rz 180 deg; joints [-9.569, -44.566, 113.769, 169.777, 69.505, -176.387]
  MoveL 4276 to (182.84, 230.28, -10) mm, rotated rx 180 ry 0 rz 180 deg; joints [-9.39, -44.559, 113.744, 169.967, 69.476, -176.451]
  MoveL 4277 to (184.22, 226.06, -10) mm, rotated rx -180 ry 0 rz -180 deg; joints [-9.212, -44.546, 113.699, 170.155, 69.435, -176.512]
  MoveL 4278 to (185.87, 221.93, -10) mm, rotated rx 180 ry 0 rz 180 deg; joints [-9.036, -44.527, 113.636, 170.34, 69.38, -176.57]
  MoveL 4279 to (187.78, 217.92, -10) mm, rotated rx -180 ry 0 rz 180 deg; joints [-8.863, -44.503, 113.555, 170.52, 69.314, -176.624]
  MoveL 4280 to (189.94, 214.04, -10) mm, rotated rx 180 ry 0 rz 180 deg; joints [-8.695, -44.473, 113.455, 170.696, 69.235, -176.676]
  MoveL 4281 to (192.34, 210.31, -10) mm, rotated rx -180 ry 0 rz -180 deg; joints [-8.531, -44.438, 113.338, 170.866, 69.144, -176.724]
  MoveL 4282 to (194.98, 206.73, -10) mm, rotated rx 180 ry 0 rz 180 deg; joints [-8.372, -44.398, 113.203, 171.03, 69.041, -176.768]
  MoveL 4283 to (197.83, 203.33, -10) mm, rotated rx 180 ry 0 rz 180 deg; joints [-8.22, -44.353, 113.052, 171.187, 68.928, -176.809]
  MoveL 4284 to (200.9, 200.11, -10) mm, rotated rx 180 ry 0 rz 180 deg; joints [-8.074, -44.303, 112.885, 171.336, 68.805, -176.846]
  MoveL 4285 to (204.16, 197.1, -10) mm, rotated rx 180 ry 0 rz 180 deg; joints [-7.936, -44.248, 112.702, 171.476, 68.671, -176.88]
  MoveL 4286 to (207.61, 194.3, -10) mm, rotated rx 180 ry 0 rz -180 deg; joints [-7.806, -44.188, 112.505, 171.608, 68.528, -176.909]
  MoveL 4287 to (211.23, 191.72, -10) mm, rotated rx -180 ry 0 rz 180 deg; joints [-7.684, -44.124, 112.294, 171.73, 68.376, -176.934]
  MoveL 4288 to (215, 189.38, -10) mm, rotated rx -180 ry 0 rz -180 deg; joints [-7.572, -44.056, 112.071, 171.842, 68.217, -176.955]
  MoveL 4289 to (218.92, 187.28, -10) mm, rotated rx 180 ry 0 rz 180 deg; joints [-7.468, -43.984, 111.835, 171.944, 68.049, -176.971]
  MoveL 4290 to (222.96, 185.44, -10) mm, rotated rx 180 ry 0 rz 180 deg; joints [-7.375, -43.908, 111.589, 172.035, 67.876, -176.984]
  MoveL 4291 to (227.11, 183.85, -10) mm, rotated rx 180 ry 0 rz 180 deg; joints [-7.292, -43.829, 111.333, 172.115, 67.696, -176.991]
  MoveL 4292 to (231.35, 182.53, -10) mm, rotated rx 180 ry 0 rz -180 deg; joints [-7.219, -43.746, 111.068, 172.183, 67.512, -176.994]
  MoveL 4293 to (235.66, 181.48, -10) mm, rotated rx -180 ry 0 rz -180 deg; joints [-7.157, -43.661, 110.796, 172.24, 67.323, -176.993]
  MoveL 4294 to (240.04, 180.71, -10) mm, rotated rx -180 ry 0 rz -180 deg; joints [-7.105, -43.573, 110.516, 172.285, 67.131, -176.986]
  MoveL 4295 to (244.45, 180.22, -10) mm, rotated rx 180 ry 0 rz 180 deg; joints [-7.065, -43.483, 110.232, 172.318, 66.935, -176.975]
  MoveL 4296 to (248.89, 180.01, -10) mm, rotated rx -180 ry 0 rz -180 deg; joints [-7.035, -43.391, 109.943, 172.338, 66.738, -176.959]
  MoveL 4297 to (253.33, 180.08, -10) mm, rotated rx -180 ry 0 rz -180 deg; joints [-7.017, -43.298, 109.651, 172.347, 66.54, -176.938]
  MoveL 4298 to (257.76, 180.43, -10) mm, rotated rx -180 ry 0 rz -180 deg; joints [-7.01, -43.204, 109.357, 172.344, 66.342, -176.912]
  MoveL 4299 to (262.16, 181.06, -10) mm, rotated rx -180 ry 0 rz -180 deg; joints [-7.013, -43.108, 109.062, 172.328, 66.144, -176.882]
  MoveL 4300 to (266.5, 181.97, -10) mm, rotated rx 180 ry 0 rz -180 deg; joints [-7.027, -43.013, 108.767, 172.301, 65.948, -176.846]
  MoveL 4301 to (270.78, 183.16, -10) mm, rotated rx -180 ry 0 rz 180 deg; joints [-7.052, -42.918, 108.475, 172.261, 65.754, -176.806]
  MoveL 4302 to (274.98, 184.61, -10) mm, rotated rx 180 ry 0 rz 180 deg; joints [-7.088, -42.823, 108.185, 172.21, 65.563, -176.761]
  MoveL 4303 to (279.08, 186.33, -10) mm, rotated rx 180 ry 0 rz 180 deg; joints [-7.134, -42.729, 107.899, 172.148, 65.375, -176.711]
  MoveL 4304 to (283.06, 188.3, -10) mm, rotated rx -180 ry 0 rz 180 deg; joints [-7.189, -42.636, 107.617, 172.075, 65.192, -176.657]
  MoveL 4305 to (286.91, 190.52, -10) mm, rotated rx 180 ry 0 rz 180 deg; joints [-7.255, -42.545, 107.343, 171.991, 65.014, -176.599]
  MoveL 4306 to (290.6, 192.98, -10) mm, rotated rx 180 ry 0 rz -180 deg; joints [-7.33, -42.456, 107.075, 171.897, 64.841, -176.536]
  MoveL 4307 to (294.14, 195.67, -10) mm, rotated rx 180 ry 0 rz 180 deg; joints [-7.413, -42.369, 106.816, 171.793, 64.676, -176.47]
  MoveL 4308 to (297.5, 198.58, -10) mm, rotated rx 180 ry 0 rz -180 deg; joints [-7.506, -42.285, 106.566, 171.68, 64.517, -176.4]
  MoveL 4309 to (300.66, 201.69, -10) mm, rotated rx 180 ry 0 rz 180 deg; joints [-7.606, -42.204, 106.326, 171.558, 64.366, -176.326]
  MoveL 4310 to (303.62, 205, -10) mm, rotated rx 180 ry 0 rz 180 deg; joints [-7.715, -42.127, 106.097, 171.427, 64.223, -176.249]
  MoveL 4311 to (306.37, 208.5, -10) mm, rotated rx -180 ry 0 rz 180 deg; joints [-7.83, -42.054, 105.881, 171.288, 64.089, -176.169]
  MoveL 4312 to (308.89, 212.16, -10) mm, rotated rx -180 ry 0 rz -180 deg; joints [-7.953, -41.984, 105.677, 171.142, 63.965, -176.087]
  MoveL 4313 to (311.17, 215.97, -10) mm, rotated rx -180 ry 0 rz -180 deg; joints [-8.082, -41.92, 105.488, 170.989, 63.85, -176.002]
  MoveL 4314 to (313.2, 219.91, -10) mm, rotated rx 180 ry 0 rz -180 deg; joints [-8.217, -41.86, 105.312, 170.83, 63.746, -175.916]
  MoveL 4315 to (314.99, 223.98, -10) mm, rotated rx 180 ry 0 rz 180 deg; joints [-8.357, -41.805, 105.152, 170.666, 63.652, -175.828]
  MoveL 4316 to (316.51, 228.16, -10) mm, rotated rx 180 ry 0 rz -180 deg; joints [-8.502, -41.756, 105.008, 170.496, 63.57, -175.739]
  MoveL 4317 to (317.76, 232.42, -10) mm, rotated rx 180 ry 0 rz -180 deg; joints [-8.652, -41.712, 104.88, 170.323, 63.498, -175.649]
  MoveL 4318 to (318.74, 236.75, -10) mm, rotated rx -180 ry 0 rz -180 deg; joints [-8.805, -41.673, 104.769, 170.146, 63.438, -175.559]
  MoveL 4319 to (319.44, 241.14, -10) mm, rotated rx -180 ry 0 rz -180 deg; joints [-8.962, -41.641, 104.676, 169.966, 63.39, -175.469]
  MoveL 4320 to (319.86, 245.56, -10) mm, rotated rx 180 ry 0 rz 180 deg; joints [-9.121, -41.615, 104.6, 169.785, 63.353, -175.379]
  MoveL 4321 to (320, 250, -10) mm, rotated rx -180 ry 0 rz -180 deg; joints [-9.282, -41.595, 104.541, 169.601, 63.329, -175.291]
  MoveL 4322 to (308, 250, -10) mm, rotated rx 180 ry 0 rz 180 deg; joints [-9.354, -41.873, 105.35, 169.569, 63.857, -175.363]
  MoveL 4323 to (307.88, 253.68, -10) mm, rotated rx 180 ry 0 rz 180 deg; joints [-9.49, -41.861, 105.317, 169.416, 63.846, -175.292]
  MoveL 4324 to (307.53, 257.34, -10) mm, rotated rx -180 ry 0 rz 180 deg; joints [-9.626, -41.855, 105.299, 169.263, 63.846, -175.222]
  MoveL 4325 to (306.95, 260.98, -10) mm, rotated rx 180 ry 0 rz 180 deg; joints [-9.764, -41.854, 105.296, 169.111, 63.856, -175.155]
  MoveL 4326 to (306.14, 264.57, -10) mm, rotated rx 180 ry 0 rz -180 deg; joints [-9.9, -41.859, 105.309, 168.96, 63.876, -175.09]
  MoveL 4327 to (305.1, 268.1, -10) mm, rotated rx -180 ry 0 rz -180 deg; joints [-10.037, -41.868, 105.337, 168.81, 63.905, -175.027]
  MoveL 4328 to (303.85, 271.56, -10) mm, rotated rx -180 ry 0 rz -180 deg; joints [-10.172, -41.883, 105.38, 168.663, 63.945, -174.967]
  MoveL 4329 to (302.37, 274.93, -10) mm, rotated rx 180 ry 0 rz -180 deg; joints [-10.305, -41.903, 105.438, 168.519, 63.994, -174.911]
  MoveL 4330 to (300.68, 278.2, -10) mm, rotated rx 180 ry 0 rz 180 deg; joints [-10.436, -41.928, 105.51, 168.378, 64.053, -174.858]
  MoveL 4331 to (298.79, 281.36, -10) mm, rotated rx -180 ry 0 rz -180 deg; joints [-10.565, -41.957, 105.598, 168.241, 64.121, -174.809]
  MoveL 4332 to (296.71, 284.39, -10) mm, rotated rx 180 ry 0 rz 180 deg; joints [-10.691, -41.992, 105.699, 168.109, 64.198, -174.763]
  MoveL 4333 to (294.43, 287.28, -10) mm, rotated rx -180 ry 0 rz 180 deg; joints [-10.813, -42.031, 105.814, 167.981, 64.283, -174.722]
  MoveL 4334 to (291.98, 290.02, -10) mm, rotated rx 180 ry 0 rz 180 deg; joints [-10.931, -42.075, 105.943, 167.859, 64.377, -174.685]
  MoveL 4335 to (289.35, 292.61, -10) mm, rotated rx -180 ry 0 rz -180 deg; joints [-11.045, -42.122, 106.084, 167.743, 64.479, -174.653]
  MoveL 4336 to (286.57, 295.02, -10) mm, rotated rx 180 ry 0 rz 180 deg; joints [-11.154, -42.174, 106.237, 167.633, 64.588, -174.625]
  MoveL 4337 to (283.64, 297.25, -10) mm, rotated rx 180 ry 0 rz 180 deg; joints [-11.257, -42.23, 106.402, 167.53, 64.705, -174.602]
  MoveL 4338 to (280.58, 299.28, -10) mm, rotated rx -180 ry 0 rz -180 deg; joints [-11.355, -42.289, 106.578, 167.435, 64.828, -174.584]
  MoveL 4339 to (277.39, 301.12, -10) mm, rotated rx 180 ry 0 rz 180 deg; joints [-11.447, -42.352, 106.764, 167.346, 64.957, -174.571]
  MoveL 4340 to (274.09, 302.76, -10) mm, rotated rx -180 ry 0 rz -180 deg; joints [-11.533, -42.417, 106.96, 167.266, 65.092, -174.563]
  MoveL 4341 to (270.7, 304.18, -10) mm, rotated rx -180 ry 0 rz 180 deg; joints [-11.611, -42.486, 107.165, 167.194, 65.233, -174.56]
  MoveL 4342 to (267.22, 305.38, -10) mm, rotated rx -180 ry 0 rz -180 deg; joints [-11.682, -42.556, 107.378, 167.13, 65.378, -174.562]
  MoveL 4343 to (263.67, 306.37, -10) mm, rotated rx 180 ry 0 rz 180 deg; joints [-11.746, -42.629, 107.597, 167.075, 65.527, -174.569]
  MoveL 4344 to (260.07, 307.12, -10) mm, rotated rx -180 ry 0 rz -180 deg; joints [-11.803, -42.704, 107.823, 167.029, 65.68, -174.581]
  MoveL 4345 to (256.43, 307.64, -10) mm, rotated rx 180 ry 0 rz 180 deg; joints [-11.851, -42.78, 108.055, 166.992, 65.836, -174.598]
  MoveL 4346 to (252.76, 307.93, -10) mm, rotated rx 180 ry 0 rz -180 deg; joints [-11.89, -42.857, 108.291, 166.965, 65.994, -174.619]
  MoveL 4347 to (249.08, 307.99, -10) mm, rotated rx -180 ry 0 rz 180 deg; joints [-11.922, -42.936, 108.53, 166.947, 66.154, -174.645]
  MoveL 4348 to (245.4, 307.82, -10) mm, rotated rx -180 ry 0 rz -180 deg; joints [-11.944, -43.015, 108.772, 166.938, 66.315, -174.676]
  MoveL 4349 to (241.75, 307.41, -10) mm, rotated rx -180 ry 0 rz -180 deg; joints [-11.958, -43.094, 109.016, 166.94, 66.477, -174.71]
  MoveL 4350 to (238.12, 306.77, -10) mm, rotated rx -180 ry 0 rz 180 deg; joints [-11.963, -43.172, 109.26, 166.95, 66.638, -174.749]
  MoveL 4351 to (234.54, 305.9, -10) mm, rotated rx -180 ry 0 rz -180 deg; joints [-11.959, -43.251, 109.504, 166.971, 66.799, -174.791]
  MoveL 4352 to (231.03, 304.81, -10) mm, rotated rx 180 ry 0 rz 180 deg; joints [-11.946, -43.329, 109.747, 167.001, 66.958, -174.837]
  MoveL 4353 to (227.59, 303.5, -10) mm, rotated rx -180 ry 0 rz -180 deg; joints [-11.923, -43.405, 109.987, 167.041, 67.116, -174.887]
  MoveL 4354 to (224.24, 301.97, -10) mm, rotated rx 180 ry 0 rz 180 deg; joints [-11.892, -43.481, 110.224, 167.09, 67.271, -174.939]
  MoveL 4355 to (221, 300.23, -10) mm, rotated rx 180 ry 0 rz 180 deg; joints [-11.851, -43.554, 110.457, 167.149, 67.422, -174.994]
  MoveL 4356 to (217.87, 298.29, -10) mm, rotated rx -180 ry 0 rz -180 deg; joints [-11.802, -43.626, 110.684, 167.216, 67.57, -175.052]
  MoveL 4357 to (214.87, 296.15, -10) mm, rotated rx -180 ry 0 rz 180 deg; joints [-11.744, -43.695, 110.906, 167.293, 67.714, -175.112]
  MoveL 4358 to (212.02, 293.83, -10) mm, rotated rx 180 ry 0 rz 180 deg; joints [-11.677, -43.762, 111.12, 167.378, 67.852, -175.174]
  MoveL 4359 to (209.31, 291.34, -10) mm, rotated rx 180 ry 0 rz 180 deg; joints [-11.602, -43.827, 111.327, 167.471, 67.984, -175.238]
  MoveL 4360 to (206.77, 288.67, -10) mm, rotated rx 180 ry 0 rz -180 deg; joints [-11.519, -43.888, 111.525, 167.572, 68.111, -175.303]
  MoveL 4361 to (204.41, 285.85, -10) mm, rotated rx -180 ry 0 rz -180 deg; joints [-11.428, -43.946, 111.713, 167.681, 68.231, -175.37]
  MoveL 4362 to (202.23, 282.89, -10) mm, rotated rx -180 ry 0 rz 180 deg; joints [-11.33, -44.001, 111.891, 167.797, 68.343, -175.437]
  MoveL 4363 to (200.24, 279.79, -10) mm, rotated rx -180 ry 0 rz 180 deg; joints [-11.224, -44.052, 112.058, 167.92, 68.448, -175.505]
  MoveL 4364 to (198.45, 276.58, -10) mm, rotated rx 180 ry 0 rz 180 deg; joints [-11.112, -44.099, 112.213, 168.049, 68.544, -175.573]
  MoveL 4365 to (196.87, 273.25, -10) mm, rotated rx 180 ry 0 rz 180 deg; joints [-10.994, -44.143, 112.356, 168.183, 68.632, -175.641]
  MoveL 4366 to (195.5, 269.84, -10) mm, rotated rx 180 ry 0 rz -180 deg; joints [-10.87, -44.182, 112.485, 168.323, 68.711, -175.709]
  MoveL 4367 to (194.35, 266.34, -10) mm, rotated rx 180 ry 0 rz 180 deg; joints [-10.741, -44.217, 112.601, 168.467, 68.781, -175.776]
  MoveL 4368 to (193.43, 262.78, -10) mm, rotated rx 180 ry 0 rz 180 deg; joints [-10.608, -44.248, 112.703, 168.616, 68.841, -175.843]
  MoveL 4369 to (192.73, 259.16, -10) mm, rotated rx 180 ry 0 rz -180 deg; joints [-10.47, -44.274, 112.79, 168.767, 68.891, -175.909]
  MoveL 4370 to (192.26, 255.51, -10) mm, rotated rx 180 ry 0 rz -180 deg; joints [-10.329, -44.296, 112.863, 168.922, 68.931, -175.974]
  MoveL 4371 to (192.03, 251.84, -10) mm, rotated rx -180 ry 0 rz 180 deg; joints [-10.185, -44.314, 112.92, 169.078, 68.96, -176.037]
  MoveL 4372 to (192.03, 248.16, -10) mm, rotated rx 180 ry 0 rz -180 deg; joints [-10.04, -44.326, 112.962, 169.236, 68.979, -176.099]
  MoveL 4373 to (192.26, 244.49, -10) mm, rotated rx -180 ry 0 rz -180 deg; joints [-9.892, -44.334, 112.988, 169.395, 68.987, -176.159]
  MoveL 4374 to (192.73, 240.84, -10) mm, rotated rx -180 ry 0 rz 180 deg; joints [-9.744, -44.337, 112.999, 169.554, 68.984, -176.217]
  MoveL 4375 to (193.43, 237.22, -10) mm, rotated rx 180 ry 0 rz 180 deg; joints [-9.596, -44.336, 112.994, 169.712, 68.971, -176.273]
  MoveL 4376 to (194.35, 233.66, -10) mm, rotated rx 180 ry 0 rz 180 deg; joints [-9.448, -44.329, 112.973, 169.869, 68.947, -176.327]
  MoveL 4377 to (195.5, 230.16, -10) mm, rotated rx -180 ry 0 rz -180 deg; joints [-9.302, -44.318, 112.936, 170.024, 68.913, -176.379]
  MoveL 4378 to (196.87, 226.75, -10) mm, rotated rx 180 ry 0 rz 180 deg; joints [-9.158, -44.303, 112.884, 170.176, 68.868, -176.428]
  MoveL 4379 to (198.45, 223.42, -10) mm, rotated rx 180 ry 0 rz -180 deg; joints [-9.016, -44.282, 112.817, 170.325, 68.813, -176.474]
  MoveL 4380 to (200.24, 220.21, -10) mm, rotated rx 180 ry 0 rz -180 deg; joints [-8.877, -44.258, 112.735, 170.47, 68.748, -176.518]
  MoveL 4381 to (202.23, 217.11, -10) mm, rotated rx 180 ry 0 rz -180 deg; joints [-8.742, -44.228, 112.638, 170.61, 68.673, -176.558]
  MoveL 4382 to (204.41, 214.15, -10) mm, rotated rx 180 ry 0 rz 180 deg; joints [-8.611, -44.195, 112.527, 170.745, 68.588, -176.596]
  MoveL 4383 to (206.77, 211.33, -10) mm, rotated rx 180 ry 0 rz 180 deg; joints [-8.486, -44.157, 112.402, 170.874, 68.495, -176.63]
  MoveL 4384 to (209.31, 208.66, -10) mm, rotated rx -180 ry 0 rz 180 deg; joints [-8.365, -44.115, 112.264, 170.997, 68.393, -176.661]
  MoveL 4385 to (212.02, 206.17, -10) mm, rotated rx -180 ry 0 rz 180 deg; joints [-8.251, -44.069, 112.113, 171.114, 68.283, -176.689]
  MoveL 4386 to (214.87, 203.85, -10) mm, rotated rx 180 ry 0 rz -180 deg; joints [-8.143, -44.019, 111.95, 171.223, 68.165, -176.713]
  MoveL 4387 to (217.87, 201.71, -10) mm, rotated rx 180 ry 0 rz 180 deg; joints [-8.042, -43.965, 111.776, 171.324, 68.04, -176.734]
  MoveL 4388 to (221, 199.77, -10) mm, rotated rx -180 ry 0 rz -180 deg; joints [-7.949, -43.908, 111.591, 171.417, 67.908, -176.751]
  MoveL 4389 to (224.24, 198.03, -10) mm, rotated rx -180 ry 0 rz -180 deg; joints [-7.863, -43.848, 111.396, 171.501, 67.771, -176.764]
  MoveL 4390 to (227.59, 196.5, -10) mm, rotated rx 180 ry 0 rz 180 deg; joints [-7.785, -43.785, 111.193, 171.577, 67.627, -176.774]
  MoveL 4391 to (231.03, 195.19, -10) mm, rotated rx -180 ry 0 rz -180 deg; joints [-7.715, -43.719, 110.981, 171.643, 67.479, -176.78]
  MoveL 4392 to (234.54, 194.1, -10) mm, rotated rx -180 ry 0 rz 180 deg; joints [-7.654, -43.65, 110.762, 171.7, 67.327, -176.781]
  MoveL 4393 to (238.12, 193.23, -10) mm, rotated rx -180 ry 0 rz -180 deg; joints [-7.602, -43.579, 110.536, 171.748, 67.171, -176.779]
  MoveL 4394 to (241.75, 192.59, -10) mm, rotated rx 180 ry 0 rz 180 deg; joints [-7.558, -43.506, 110.305, 171.785, 67.012, -176.773]
  MoveL 4395 to (245.4, 192.18, -10) mm, rotated rx 180 ry 0 rz 180 deg; joints [-7.524, -43.431, 110.069, 171.813, 66.851, -176.763]
  MoveL 4396 to (249.08, 192.01, -10) mm, rotated rx -180 ry 0 rz 180 deg; joints [-7.498, -43.355, 109.83, 171.831, 66.688, -176.749]
  MoveL 4397 to (252.76, 192.07, -10) mm, rotated rx -180 ry 0 rz -180 deg; joints [-7.482, -43.278, 109.588, 171.839, 66.524, -176.73]
  MoveL 4398 to (256.43, 192.36, -10) mm, rotated rx -180 ry 0 rz 180 deg; joints [-7.475, -43.2, 109.344, 171.836, 66.36, -176.708]
  MoveL 4399 to (260.07, 192.88, -10) mm, rotated rx -180 ry 0 rz 180 deg; joints [-7.476, -43.121, 109.1, 171.824, 66.196, -176.681]
  MoveL 4400 to (263.67, 193.63, -10) mm, rotated rx 180 ry 0 rz 180 deg; joints [-7.487, -43.042, 108.856, 171.802, 66.034, -176.651]
  MoveL 4401 to (267.22, 194.62, -10) mm, rotated rx -180 ry 0 rz -180 deg; joints [-7.507, -42.963, 108.613, 171.77, 65.873, -176.616]
  MoveL 4402 to (270.7, 195.82, -10) mm, rotated rx -180 ry 0 rz -180 deg; joints [-7.535, -42.884, 108.373, 171.729, 65.714, -176.578]
  MoveL 4403 to (274.09, 197.24, -10) mm, rotated rx -180 ry 0 rz 180 deg; joints [-7.572, -42.807, 108.136, 171.678, 65.558, -176.536]
  MoveL 4404 to (277.39, 198.88, -10) mm, rotated rx -180 ry 0 rz -180 deg; joints [-7.617, -42.73, 107.903, 171.618, 65.406, -176.491]
  MoveL 4405 to (280.58, 200.72, -10) mm, rotated rx 180 ry 0 rz 180 deg; joints [-7.671, -42.655, 107.675, 171.549, 65.259, -176.442]
  MoveL 4406 to (283.64, 202.75, -10) mm, rotated rx -180 ry 0 rz 180 deg; joints [-7.732, -42.581, 107.453, 171.471, 65.116, -176.389]
  MoveL 4407 to (286.57, 204.98, -10) mm, rotated rx 180 ry 0 rz 180 deg; joints [-7.801, -42.51, 107.237, 171.385, 64.978, -176.334]
  MoveL 4408 to (289.35, 207.39, -10) mm, rotated rx -180 ry 0 rz 180 deg; joints [-7.877, -42.441, 107.03, 171.292, 64.846, -176.275]
  MoveL 4409 to (291.98, 209.98, -10) mm, rotated rx 180 ry 0 rz -180 deg; joints [-7.96, -42.374, 106.831, 171.191, 64.721, -176.214]
  MoveL 4410 to (294.43, 212.72, -10) mm, rotated rx -180 ry 0 rz 180 deg; joints [-8.05, -42.31, 106.641, 171.083, 64.602, -176.15]
